# B&R Automation Studio project MotionTestBenchMaster (part 6)

#### SwChg.st - Monitor and write into the user logger the canges of the software objects
```iecst
(********************************************************************
 * COPYRIGHT --
 ********************************************************************
 * Library: Powertoys
 * File: swChg.st
 * Author: Massimo Gibertini
 * Created: August 07, 2014
 ********************************************************************
 * Implementation of library Powertoys
 ********************************************************************)

(* Monitor and write into the user logger the canges of the software objects *)
FUNCTION_BLOCK SwChg

	IF (enable = TRUE) THEN
		customEntry.logLevel 		:= logLevel;
		waitWrite.PT				:= T#10m;

		CASE step OF

			0:
				(* Getting the software list *)
				busy			:= TRUE;
				searching		:= FALSE;
				writingLog		:= FALSE;
				waiting			:= FALSE;
				scan			:= TRUE;
				error			:= FALSE;
				errorID			:= ERR_FUB_BUSY;

				CASE substep OF

					0:
						memset(ADR(tempModule),0,SIZEOF(tempModule));
						memset(ADR(iActList),0,SIZEOF(iActList));
						memset(ADR(iOldList),0,SIZEOF(iOldList));

						(* Checking if the swList temporary data object exist in the userRam or not*)
						datObjInfo_0.pName 	:= ADR(swListTempDataObjName);
						datObjInfo_0.enable	:= TRUE;
						substep 			:= 1;

					1:
						datObjInfo_0();
						IF (datObjInfo_0.status = doERR_MODULNOTFOUND) THEN
							(* Temporary data object not found *)
							swListTempID	:= 0;
							substep			:= 5;
						ELSIF (datObjInfo_0.status = ERR_OK) THEN
							(* Data object found *)
							swListTempID	:= datObjInfo_0.ident;
							//substep			:= 2;
							substep			:= 5;
						ELSIF (datObjInfo_0.status <> ERR_OK) AND (datObjInfo_0.status <> doERR_MODULNOTFOUND) AND (datObjInfo_0.status <> ERR_FUB_BUSY) THEN
							errorID			:= datObjInfo_0.status;
							errorStep		:= step;
							errorSubStep	:= substep;
							step 			:= 200;
							substep			:= 0;
						END_IF;

					2:
						datObjInfo_0.enable	:= FALSE;
						datObjInfo_0();
						IF (datObjInfo_0.status = ERR_FUB_ENABLE_FALSE) THEN
							substep			:= 3;
						END_IF;

					3:
						(* Delete the temporary data object *)
						datObjDelete_0.ident	:= swListTempID;
						datObjDelete_0.enable	:= TRUE;
						substep					:= 4;

					4:
						datObjDelete_0();
						IF (datObjDelete_0.status = ERR_OK) THEN
							substep			:= 5;
							swListTempID	:= 0;
						ELSIF (datObjDelete_0.status <> ERR_OK) AND (datObjDelete_0.status <> ERR_FUB_BUSY) THEN
							errorID			:= datObjDelete_0.status;
							errorStep		:= step;
							errorSubStep	:= substep;
							step 			:= 200;
							substep			:= 0;
						END_IF;

					5:
						(* Disable fub *)
						datObjDelete_0.enable	:= FALSE;
						datObjDelete_0();
						datObjInfo_0.enable	:= FALSE;
						datObjInfo_0();
						IF (datObjDelete_0.status = ERR_FUB_ENABLE_FALSE) AND (datObjInfo_0.status = ERR_FUB_ENABLE_FALSE) THEN
							substep				:= 6;
						END_IF;

					6:
						(* temporary data object not present or deleted *)
						(* Checking if the swList data object exist or not *)
						datObjInfo_0.pName 	:= ADR(swListDatObjName);
						datObjInfo_0.enable	:= TRUE;
						datObjInfo_0();
						IF (datObjInfo_0.status <> ERR_FUB_BUSY) AND (datObjInfo_0.status <> ERR_FUB_ENABLE_FALSE) THEN
							substep := 7;
						END_IF;

					7:
						datObjInfo_0();
						IF (datObjInfo_0.status = doERR_MODULNOTFOUND) THEN
							(* Data object not found *)
							swListID		:= 0;
							substep			:= 100;
						ELSIF (datObjInfo_0.status = doERR_CHECKSUM_WARNING) THEN
							swListID		:= datObjInfo_0.ident;
							substep			:= 10;
						ELSIF (datObjInfo_0.status = ERR_OK) THEN
							(* Data object found *)
							swListID		:= datObjInfo_0.ident;
							IF (swListTempID = 0) THEN
								substep			:= 50;
							ELSE
								substep 		:= 150;
							END_IF;

						ELSIF (datObjInfo_0.status <> ERR_OK) AND (datObjInfo_0.status <> doERR_CHECKSUM_WARNING) AND (datObjInfo_0.status <> doERR_MODULNOTFOUND) AND (datObjInfo_0.status <> ERR_FUB_BUSY) THEN
							errorID			:= datObjInfo_0.status;
							errorStep		:= step;
							errorSubStep	:= substep;
							step 			:= 200;
							substep			:= 0;
						END_IF;

					(* Data object damaged, deleting *)
					10:
						datObjInfo_0.enable	:= FALSE;
						datObjInfo_0();
						IF (datObjInfo_0.status = ERR_FUB_ENABLE_FALSE) THEN
							substep			:= 11;
						END_IF;

					11:
						datObjDelete_0.ident	:= swListID;
						datObjDelete_0.enable	:= TRUE;
						datObjDelete_0();
						IF (datObjDelete_0.status <> ERR_FUB_BUSY) AND (datObjDelete_0.status <> ERR_FUB_ENABLE_FALSE) THEN
							substep 				:= 12;
						END_IF;

					12:
						datObjDelete_0();
						IF (datObjDelete_0.status = ERR_OK) THEN
							substep				:= 13;
						ELSIF (datObjDelete_0.status <> ERR_OK) AND (datObjDelete_0.status <> ERR_FUB_BUSY) THEN
							errorID				:= datObjDelete_0.status;
							errorStep			:= step;
							errorSubStep		:= substep;
							step 				:= 200;
							substep				:= 0;
						END_IF;

					13:
						datObjDelete_0.enable	:= FALSE;
						datObjDelete_0();
						IF (datObjDelete_0.status = ERR_FUB_ENABLE_FALSE) THEN
							(* No existing data object *)
							substep 			:= 100;
							swListID 			:= 0;
						END_IF;

					50:
						(* swList data object present, copy to DRam *)
						datObjInfo_0.enable			:= FALSE;
						datObjCopy_0.ident 			:= swListID;
						datObjCopy_0.pNameTarget 	:= ADR(swListTempDataObjName);
						datObjCopy_0.MemTypeTarget	:= doTEMP;
						datObjCopy_0.enable			:= TRUE;
						datObjCopy_0();
						substep := 51;

					51:
						datObjCopy_0();
						IF (datObjCopy_0.status = ERR_OK) THEN
							substep 				:= 52;
							swListTempID			:= datObjCopy_0.identNew;
						ELSIF (datObjCopy_0.status <> ERR_OK) AND (datObjCopy_0.status <> ERR_FUB_BUSY) THEN
							errorID					:= datObjCopy_0.status;
							errorStep				:= step;
							errorSubStep			:= substep;
							step 					:= 200;
							substep					:= 0;
						END_IF;

					52:
						datObjCopy_0.enable			:= FALSE;
						datObjCopy_0();
						IF (datObjCopy_0.status = ERR_FUB_ENABLE_FALSE) THEN
							(* Temporary Data object recovered succesfully *)
							substep					:= 150;

						END_IF;

					100:
						(* Creating the temporary data object*)
						IF (swListTempID = 0) THEN
							datObjInfo_0.enable		:= FALSE;
							datObjCreate_0.grp		:= 0;
							datObjCreate_0.pName	:= ADR(swListTempDataObjName);
							datObjCreate_0.len		:= SIZEOF(iActList);
							datObjCreate_0.MemType	:= doTEMP;
							datObjCreate_0.Option	:= doNO_CS;
							datObjCreate_0.pCpyData	:= ADR(iActList);
							datObjCreate_0.enable	:= TRUE;
							datObjCreate_0();
							substep					:= 101;
						ELSE
							substep					:= 110;
						END_IF;

					101:
						datObjCreate_0();
						IF (datObjCreate_0.status = ERR_OK) THEN
							substep				:= 102;
							swListTempID		:= datObjCreate_0.ident;
							newSwListT			:= TRUE;
						ELSIF (datObjCreate_0.status <> ERR_OK) AND (datObjCreate_0.status <> ERR_FUB_BUSY) THEN
							errorID				:= datObjCreate_0.status;
							errorStep			:= step;
							errorSubStep		:= substep;
							step 				:= 200;
							substep				:= 0;
						END_IF;

					102:
						datObjCreate_0.enable	:= FALSE;
						datObjCreate_0();
						IF (datObjCreate_0.status = ERR_FUB_ENABLE_FALSE) THEN
							substep				:= 110;

						END_IF;

					110:
						(* Creating the cf data object*)
						datObjCreate_0.grp		:= 0;
						datObjCreate_0.pName	:= ADR(swListDatObjName);
						datObjCreate_0.len		:= SIZEOF(iOldList);
						datObjCreate_0.MemType	:= doUSRROM;
						datObjCreate_0.Option	:= 0;
						datObjCreate_0.pCpyData	:= ADR(iOldList);
						datObjCreate_0.enable	:= TRUE;
						substep					:= 112;

					112:
						datObjCreate_0();
						IF (datObjCreate_0.status = ERR_OK) THEN
							substep					:= 113;
							swListID				:= datObjCreate_0.ident;
							datObjCreate_0.enable	:= FALSE;
						ELSIF (datObjCreate_0.status <> ERR_OK) AND (datObjCreate_0.status <> ERR_FUB_BUSY) THEN
							errorID					:= datObjCreate_0.status;
							errorStep				:= step;
							errorSubStep			:= substep;
							step 					:= 200;
							substep					:= 0;
						END_IF;

					113:
						datObjCreate_0.enable		:= FALSE;
						datObjCreate_0();
						IF (datObjCreate_0.status = ERR_FUB_ENABLE_FALSE) AND newSwListT THEN
							substep					:= 200;
							oldListElements			:= 0;
						ELSIF (datObjCreate_0.status = ERR_FUB_ENABLE_FALSE) AND NOT (newSwListT) THEN
							substep					:= 150;
							oldListElements			:= 0;
						END_IF;

					150:
						(* Loading the existing temporary data object *)
						datObjRead_0.ident			:= swListTempID;
						datObjRead_0.Offset			:= 0;
						datObjRead_0.pDestination	:= ADR(iOldList);
						datObjRead_0.len			:= SIZEOF(iOldList);
						datObjRead_0.enable			:= TRUE;
						datObjRead_0();
						substep						:= 151;

					151:

						datObjRead_0();
						IF (datObjRead_0.status = ERR_OK) THEN
							substep					:= 152;
						ELSIF (datObjRead_0.status <> ERR_OK) AND (datObjRead_0.status <> ERR_FUB_BUSY)	THEN
							errorID					:= datObjRead_0.status;
							errorStep				:= step;
							errorSubStep			:= substep;
							step 					:= 200;
							substep					:= 0;
						END_IF;

					152:
						datObjRead_0.enable			:= FALSE;
						datObjRead_0();
						IF (datObjRead_0.status = ERR_FUB_ENABLE_FALSE) THEN
							oldListElements 		:= 0;
							substep 				:= 153;
						END_IF;

					153:
						(* Listing the number of entries in the old list *)
						memset(ADR(tempString),0,SIZEOF(tempString));
						memcpy(ADR(tempString),ADR(iOldList[oldListElements].module.name[0]),SIZEOF(iOldList[oldListElements].module.name));
						IF (tempString <> '') THEN
							oldListElements := oldListElements + 1;
						ELSE
							substep 		:= 200;
						END_IF;

					200:
						(* Cleaning the memory of the actual list *)
						(* Listing all the software objects *)
						memset(ADR(iActList),0,SIZEOF(iActList));
						mo_prev_index 	:= 16#FFFF;
						mo_index 		:= 0;
						nrChanges 		:= 0;
						substep			:= 201;

					201:
						(* Listing all the software objects element *)
						memset(ADR(tempModule), 0, SIZEOF(tempModule));
						MO_list(mo_prev_index, ADR(mo_index),ADR(tempModule));

						IF (tempModule.type <> 0) AND ((tempModule.type = CST_configOBJ)	OR
							(tempModule.type = CST_cycOBJ)		OR
							(tempModule.type = CST_fwOBJ)		OR
							(tempModule.type = CST_hwOBJ)		OR
							(tempModule.type = CST_ncOBJ)		OR
							(tempModule.type = CST_sysOBJ))		THEN

							(* Valid system object *)
							MO_ver(ADR(tempModule.name),0,ADR(iActList[nrChanges].version));
							memcpy(ADR(iActList[nrChanges].module.name[0]),ADR(tempModule.name[0]), SIZEOF(tempModule.name));

							iActList[nrChanges].module.grp		:= tempModule.grp;
							iActList[nrChanges].module.memtype	:= tempModule.memtype;
							iActList[nrChanges].module.reserve 	:= tempModule.reserve;
							iActList[nrChanges].module.state	:= tempModule.state;
							iActList[nrChanges].module.type		:= tempModule.type;

							nrChanges							:= nrChanges + 1;
							substep 							:= 202;
						ELSE
							substep 							:= 202;
						END_IF;

					202:
						(* Checking if I have finished to scan *)

						IF (mo_prev_index = mo_index) OR (nrChanges = iMaxEntries) THEN
							substep 		:= 203;
						ELSE
							mo_prev_index	:= mo_index;
							substep 		:= 201;
						END_IF;

					203:
						(* Software list complete *)
						actListElements 	:= nrChanges;
						step 				:= 1;
						substep 			:= 0;

				END_CASE;

			1:
				(* Searching for modified software objects *)
				busy			:= TRUE;
				searching		:= TRUE;
				writingLog		:= FALSE;
				waiting			:= FALSE;
				scan			:= FALSE;
				error			:= FALSE;
				errorID			:= ERR_FUB_BUSY;

				CASE substep OF
					0:
						(* Software list complete, comparing memory area *)
						IF (memcmp(ADR(iActList), ADR(iOldList), SIZEOF(iActList)) = 0) THEN

							(* No software changes *)
							substep	:= 0;
							step	:= 20;

						ELSE

							(* There are some changes *)
							substep		:= 1;
							cnt			:= 0;
							nrChanges	:= 0;
							oldSubStep	:= 0;
						END_IF;

					1:
						(* Trying to find the module in the same position of the old array *)
						(* First speed up improvement *)
						IF ((memcmp(ADR(iActList[nrChanges].module.name[0]), ADR(iOldList[nrChanges].module.name[0]), SIZEOF(iOldList[nrChanges].module.name)) = 0)
							AND (cnt < oldListElements) AND (nrChanges < actListElements)) THEN

							(* Module found *)
							IF (memcmp(ADR(iActList[nrChanges]),ADR(iOldList[nrChanges]),SIZEOF(iOldList[nrChanges])) = 0) THEN

								(* The module are the same *)
								nrChanges	:= nrChanges + 1;
								cnt			:= 0;
							ELSE

								(* The module is modified *)
								substep 	:= 10;
								step		:= 10;

							END_IF;

						ELSE
							(* Module not found *)
							substep 	:= 10;

						END_IF;

					10:
						(* Comparing the all elements of the iActList with all the elements of iOldList to find if the element exist or not *)
						IF (memcmp(ADR(iActList[nrChanges].module.name[0]), ADR(iOldList[cnt].module.name[0]), SIZEOF(iOldList[cnt].module.name)) <> 0) AND (nrChanges < actListElements) THEN
							IF (cnt < oldListElements)  THEN
								(* Module not found *)
								cnt 		:= cnt + 1;

							ELSIF (cnt >= oldListElements)  THEN

								(* New software module *)
								substep		:= 20;
								step		:= 10;
							END_IF;

						ELSIF ((memcmp(ADR(iActList[nrChanges].module.name[0]), ADR(iOldList[cnt].module.name[0]), SIZEOF(iOldList[cnt].module.name)) = 0)
								AND (cnt < oldListElements) AND (nrChanges < actListElements)) THEN

							(* Module found *)
							IF (memcmp(ADR(iActList[nrChanges]),ADR(iOldList[cnt]),SIZEOF(iOldList[cnt])) = 0) THEN

								(* The module are the same *)
								nrChanges	:= nrChanges + 1;
								cnt			:= 0;
								substep 	:= 1;
							ELSE

								(* The module is modified *)
								substep 	:= 10;
								step		:= 10;
							END_IF;

						ELSIF (nrChanges >= actListElements) THEN

							(* Search finished, checking the removed objects *)
							substep			:= 2;
							cnt 			:= 0;
							nrChanges 		:= 0;
						END_IF;

					2:
						(* Trying to find the module in the same position of the old array *)
						(* Second speed up improvement *)
						IF ((memcmp(ADR(iActList[cnt].module.name[0]), ADR(iOldList[cnt].module.name[0]), SIZEOF(iOldList[cnt].module.name)) = 0)
							AND (cnt < oldListElements) AND (nrChanges < actListElements)) THEN

							(* Module found *)
							cnt				:= cnt + 1;
							nrChanges		:= 0;

						ELSE
							(* Module not found *)
							nrChanges		:= 0;
							substep 	:= 20;
						END_IF

					20:
						(* Checking if there are any removed software object *)
						IF (memcmp(ADR(iActList[nrChanges].module.name[0]), ADR(iOldList[cnt].module.name[0]), SIZEOF(iOldList[cnt].module.name)) <> 0) AND (oldListElements <> 0) AND (cnt < oldListElements) THEN

							IF  (nrChanges < actListElements) THEN

								(* Module not found *)
								nrChanges	:= nrChanges + 1;

							ELSIF (nrChanges >= actListElements) THEN

								(* SW module removed *)
								substep 	:= 0;
								step		:= 10;
							END_IF;

						ELSIF ((memcmp(ADR(iActList[nrChanges].module.name[0]), ADR(iOldList[cnt].module.name[0]), SIZEOF(iOldList[cnt].module.name)) = 0)
							AND (cnt < oldListElements) AND (nrChanges < actListElements)) THEN

							(* Module found *)
							cnt				:= cnt + 1;
							substep 		:= 2;
							nrChanges		:= 0;

						ELSIF (cnt >= oldListElements) THEN

							(* Search finished *)
							step			:= 10;
							substep 		:= 30;
							cnt				:= 0;
							nrChanges		:= 0;
						END_IF;

				END_CASE;

			10:
				(* Writing informations into the logger and data object *)
				busy 			:= TRUE;
				searching 		:= FALSE;
				writingLog		:= TRUE;
				waiting 		:= FALSE;
				scan			:= FALSE;
				error			:= FALSE;
				errorID			:= ERR_FUB_BUSY;

				CASE substep OF

					0:
						(* Removed software module *)
						memset(ADR(tempString),0,SIZEOF(tempString));
						tempString	:= 'REMOVED SW MODULE: ';
						memcpy(ADR(tempString)+LEN(tempString),ADR(iOldList[cnt].module.name[0]), SIZEOF(iOldList[cnt].module.name));
						substep		:= 1;

					1:
						(* Writing into the logger *)
						customEntry.adr_string 		:= ADR(tempString);
						customEntry.errorNum 		:= LOG_SW_OBJ_CHG;
						writeDiff.adrCustomEntry 	:= ADR(customEntry);
						writeDiff.enable 			:= TRUE;
						substep 					:= 2;

					2:

						IF (writeDiff.done = TRUE) THEN
							substep			:= 3;
						ELSIF (writeDiff.error) THEN
							errorID			:= writeDiff.errorID;
							errorStep		:= step;
							errorSubStep	:= substep;
							step 			:= 200;
							substep			:= 0;
						END_IF;

					3:
						writeDiff.enable	:= FALSE;
						IF (writeDiff.errorID = ERR_FUB_ENABLE_FALSE) THEN
							cnt				:= cnt + 1;
							nrChanges		:= 0;
							step			:= 1;
							substep			:= 2;
						END_IF;

					10:
						(* Modified software module *)
						memset(ADR(tempString),0,SIZEOF(tempString));
						tempString	:= 'MODIFIED SW MODULE: ';
						memcpy(ADR(tempString)+LEN(tempString),ADR(iActList[nrChanges].module.name[0]), SIZEOF(iActList[nrChanges].module.name));
						substep		:= 11;

					11:
						(* Writing into the logger *)
						customEntry.adr_string 		:= ADR(tempString);
						customEntry.errorNum 		:= LOG_SW_OBJ_CHG;
						writeDiff.adrCustomEntry 	:= ADR(customEntry);
						writeDiff.enable 			:= TRUE;
						substep 					:= 12;

					12:

						IF (writeDiff.done = TRUE) THEN
							substep			:= 13;
						ELSIF (writeDiff.error) THEN
							errorID			:= writeDiff.errorID;
							errorStep		:= step;
							errorSubStep	:= substep;
							step 			:= 200;
							substep			:= 0;
						END_IF;

					13:
						writeDiff.enable	:= FALSE;
						IF (writeDiff.errorID = ERR_FUB_ENABLE_FALSE) THEN
							cnt				:= 0;
							nrChanges		:= nrChanges + 1;
							substep			:= 1;
							step			:= 1;
						END_IF;

					20:
						(* New software module *)
						memset(ADR(tempString),0,SIZEOF(tempString));
						tempString	:= 'NEW SW MODULE: ';
						memcpy(ADR(tempString)+LEN(tempString),ADR(iActList[nrChanges].module.name[0]), SIZEOF(iActList[nrChanges].module.name));
						substep		:= 21;

					21:
						(* Writing into the logger *)
						customEntry.adr_string 		:= ADR(tempString);
						customEntry.errorNum 		:= LOG_SW_OBJ_NEW;
						writeDiff.adrCustomEntry 	:= ADR(customEntry);
						writeDiff.enable 			:= TRUE;
						substep						:= 22;

					22:
						IF (writeDiff.done = TRUE) THEN
							substep			:= 23;
						ELSIF (writeDiff.error) THEN
							errorID			:= writeDiff.errorID;
							errorStep		:= step;
							errorSubStep	:= substep;
							step 			:= 200;
							substep			:= 0;
						END_IF;

					23:
						writeDiff.enable	:= FALSE;
						IF (writeDiff.errorID = ERR_FUB_ENABLE_FALSE) THEN
							cnt				:= 0;
							nrChanges		:= nrChanges + 1;
							substep			:= 1;
							step			:= 1;
						END_IF;

					30:
						(* Writing temporary data object *)
						datObjWrite_0.ident		:= swListTempID;
						datObjWrite_0.len		:= SIZEOF(iActList);
						datObjWrite_0.Offset	:= 0;
						datObjWrite_0.pSource	:= ADR(iActList);
						datObjWrite_0.enable	:= TRUE;
						datObjWrite_0();
						substep					:= 31;

					31:
						datObjWrite_0();
						IF (datObjWrite_0.status = ERR_OK) THEN
							substep 				:= 50;
							waitWrite.IN 			:= TRUE;
							datObjWrite_0.enable 	:= FALSE;
						ELSIF (datObjWrite_0.status <> ERR_OK) AND (datObjWrite_0.status <> ERR_FUB_BUSY) THEN
							errorID					:= datObjWrite_0.status;
							errorStep				:= step;
							errorSubStep			:= substep;
							step 					:= 200;
							substep					:= 0;
						END_IF;

					40:
						(* Writing cf data object *)
						datObjWrite_0.ident			:= swListID;
						datObjWrite_0.len			:= SIZEOF(iActList);
						datObjWrite_0.Offset		:= 0;
						datObjWrite_0.pSource		:= ADR(iActList);
						datObjWrite_0.enable		:= TRUE;
						datObjWrite_0();
						substep						:= 41;
					41:
						datObjWrite_0();
						IF (datObjWrite_0.status = ERR_OK) THEN
							substep 				:= 50;
							waitWrite.IN 			:= FALSE;
							datObjWrite_0.enable 	:= FALSE;
						ELSIF (datObjWrite_0.status <> ERR_OK) AND (datObjWrite_0.status <> ERR_FUB_BUSY) THEN
							errorID					:= datObjWrite_0.status;
							errorStep				:= step;
							errorSubStep			:= substep;
							step 					:= 200;
							substep					:= 0;
						END_IF;

					50:
						(* Copy the actual list into the old list *)
						memcpy(ADR(iOldList), ADR(iActList), SIZEOF(iActList));
						memset(ADR(tempString),0,SIZEOF(tempString));
						substep := 0;
						step 	:= 20;
				END_CASE;

			20:
				(* Waiting step *)
				busy 			:= TRUE;
				searching 		:= FALSE;
				writingLog		:= FALSE;
				waiting 		:= TRUE;
				scan			:= FALSE;
				error			:= FALSE;
				errorID			:= ERR_FUB_BUSY;

				CASE substep OF
					0:
						(* No software changes *)
						refresh.PT := refreshTime;
						refresh.IN := TRUE;

						IF refresh.Q THEN
							substep := 1;
						END_IF;

					1:
						(* Refresh time elapsed *)
						IF (waitWrite.Q) THEN
							step 	:= 10;
							substep := 40;
						ELSE
							refresh.IN := FALSE;
							step 	:= 0;
							substep := 152;
						END_IF;

				END_CASE;

			200:
				(* Error state resetting all the used function block *)
				writeDiff.enable		:= FALSE;
				refresh.IN 				:= FALSE;
				waitWrite.IN			:= FALSE;
				datObjWrite_0.enable	:= FALSE;
				datObjInfo_0.enable		:= FALSE;
				datObjDelete_0.enable	:= FALSE;
				datObjRead_0.enable		:= FALSE;
				datObjCreate_0.enable	:= FALSE;
				datObjCopy_0.enable		:= FALSE;

				(* Updating the status *)
				busy			:= FALSE;
				searching		:= FALSE;
				writingLog		:= FALSE;
				waiting			:= FALSE;
				scan			:= FALSE;
				error			:= TRUE;
		END_CASE;

	ELSE

		mo_prev_index 	:= 16#FFFF;
		mo_index 		:= 0;
		cnt 			:= 0;
		nrChanges 		:= 0;
		substep			:= 0;
		step			:= 0;
		errorSubStep	:= 0;
		errorStep		:= 0;
		oldSubStep		:= 0;

		oldListElements := 0;
		actListElements	:= 0;

		error			:= TRUE;
		errorID			:= ERR_FUB_ENABLE_FALSE;
		busy			:= FALSE;
		searching		:= FALSE;
		writingLog		:= FALSE;
		waiting			:= FALSE;
		scan			:= FALSE;
		newSwListT		:= FALSE;
		(* Resetting all the used function block *)
		writeDiff.enable		:= FALSE;
		refresh.IN 				:= FALSE;
		waitWrite.IN			:= FALSE;
		datObjWrite_0.enable	:= FALSE;
		datObjInfo_0.enable		:= FALSE;
		datObjDelete_0.enable	:= FALSE;
		datObjRead_0.enable		:= FALSE;
		datObjCreate_0.enable	:= FALSE;
		datObjCopy_0.enable		:= FALSE;
	END_IF;

	writeDiff();
	refresh();
	waitWrite();

END_FUNCTION_BLOCK
```

#### LogSupplyEvents.st - Write the power supply events in the specified logger
```iecst
(********************************************************************
 * COPYRIGHT -- Bernecker + Rainer
 ********************************************************************
 * Library: GenUps
 * File: LogSupplyEvents.st
 * Author: gibertinim
 * Created: March 13, 2014
 ********************************************************************
 * Implementation of library GenUps
 ********************************************************************)

(* Write the power supply events in the specified logger *)
FUNCTION_BLOCK LogSupplyEvents

	IF (enable = TRUE) THEN

		CASE step OF

			0:
				pUpsIO ACCESS (ADR_UpsIO);

				errorID 			:=	ERR_FUB_BUSY;
				busy				:=	TRUE;
				error				:=	FALSE;
				noSupply			:= TRUE;
				batteryLow			:= FALSE;
				batteryAlarm		:= FALSE;
				shutdownRequested	:= FALSE;

				IF (customLogEntry_0.errorID = ERR_FUB_ENABLE_FALSE) THEN
					(* The function block started running *)
					step := 1;
				END_IF;

			1:

				memset(ADR(data),0,SIZEOF(data));
				customLogEntry_0.adrCustomEntry	:=	ADR(data);
				memset(ADR(tempString),0,SIZEOF(tempString));
				memset(ADR(tempString2),0,SIZEOF(tempString2));

				IF (pUpsIO.shutdownAlarm = TRUE) THEN
					step := 50;
				ELSE
					step := 51;
				END_IF;

			2:
				(* Waiting for an event *)

				IF 		((pUpsIO.batteryAlarm	= TRUE)		AND	(batteryAlarm		= FALSE))	THEN
					step := 10;
				ELSIF	((pUpsIO.batteryAlarm	= FALSE)	AND	(batteryAlarm		= TRUE))	THEN
					step := 11;
				ELSIF	((pUpsIO.batteryLow		= TRUE)		AND	(batteryLow			= FALSE))	THEN
					step := 20;
				ELSIF	((pUpsIO.batteryLow		= FALSE)	AND	(batteryLow			= TRUE))	THEN
					step := 21;
				ELSIF	((pUpsIO.noPowerSupply	= TRUE)		AND (noSupply			= FALSE))	THEN
					step := 30;
				ELSIF	((pUpsIO.noPowerSupply	= FALSE)	AND (noSupply			= TRUE))	THEN
					step := 31;
				ELSIF (pUpsIO.shutdownReq		= TRUE)		AND	(shutdownRequested	= FALSE)	THEN
					step := 40;
				ELSIF(	(pUpsIO.batteryAlarm	= FALSE)	AND	(batteryAlarm		= FALSE)	AND
						(pUpsIO.batteryLow		= FALSE)	AND	(batteryLow			= FALSE)	AND
						(pUpsIO.noPowerSupply	= FALSE)	AND (noSupply			= FALSE)	AND
						(pUpsIO.shutdownReq 	= FALSE)	AND (shutdownRequested	= FALSE))	THEN
					upsStatus := ERR_OK;
				ELSIF (	(pUpsIO.shutdownReq 	= FALSE)	AND (shutdownRequested	= TRUE)) THEN
					shutdownRequested := FALSE;
				END_IF;

			10:

				customLogEntry_0.enable 		:= 	TRUE;

				data.errorNum		:= ERR_UPS_BATTERY_FAULT;
				data.adr_string		:= ADR('UPS BATTERY FAULT');
				data.logLevel		:= arEVENTLOG_SEVERITY_WARNING;
				batteryAlarm		:= TRUE;
				upsStatus			:= ERR_UPS_BATTERY_FAULT;
				(* Waiting until the log is written succesfully *)
				IF (customLogEntry_0.errorID = ERR_OK) THEN
					(* Log entry written succesfully*)
					step 					:= 101;
					customLogEntry_0.enable := 	FALSE;
				ELSIF ((customLogEntry_0.errorID <> ERR_FUB_BUSY) AND (customLogEntry_0.errorID <> ERR_OK)AND (customLogEntry_0.errorID <> ERR_FUB_ENABLE_FALSE)) THEN
					(* Error occured while saving the logger *)
					errorStep	:= 10;
					errorID		:= customLogEntry_0.errorID;
					error		:= TRUE;
					step		:= 200;
				END_IF;

			11:
				(* Battery alarm recovered *)

				customLogEntry_0.enable := 	TRUE;
				data.errorNum			:= ERR_UPS_BATTERY_OK;

				data.adr_string	:= ADR('UPS BATTERY FAULT RECOVERED');
				data.logLevel	:= arEVENTLOG_SEVERITY_INFO;
				batteryAlarm	:= FALSE;
				(* Waiting until the log is written succesfully *)

				IF (customLogEntry_0.errorID = ERR_OK) THEN
					(* Log entry written succesfully*)
					step 					:= 101;
					customLogEntry_0.enable := FALSE;
				ELSIF ((customLogEntry_0.errorID <> ERR_FUB_BUSY) AND customLogEntry_0.errorID <> ERR_OK)AND (customLogEntry_0.errorID <> ERR_FUB_ENABLE_FALSE) THEN
					(* Error occured while saving the logger *)
					errorStep	:= 11;
					errorID		:= customLogEntry_0.errorID;
					error		:= TRUE;
					step		:= 200;
				END_IF;

			20:

				(* Battery low *)

				customLogEntry_0.enable 		:= 	TRUE;
				data.errorNum		:= ERR_UPS_BATTERY_LOW;
				data.adr_string		:= ADR('UPS BATTERY LOW');
				data.logLevel		:= arEVENTLOG_SEVERITY_WARNING;
				batteryLow			:= TRUE;
				upsStatus			:= ERR_UPS_BATTERY_LOW;
				(* Waiting until the log is written succesfully *)
				IF (customLogEntry_0.errorID = ERR_OK) THEN
					(* Log entry written succesfully*)
					step 					:= 101;
					customLogEntry_0.enable := FALSE;
				ELSIF ((customLogEntry_0.errorID <> ERR_FUB_BUSY) AND (customLogEntry_0.errorID <> ERR_OK)AND (customLogEntry_0.errorID <> ERR_FUB_ENABLE_FALSE)) THEN
					(* Error occured while saving the logger *)
					errorStep	:= 20;
					errorID		:= customLogEntry_0.errorID;
					error		:= TRUE;
					step		:= 200;
				END_IF;

			21:
				(* Battery recharged *)

				customLogEntry_0.enable 		:= 	TRUE;

				data.errorNum		:= ERR_UPS_BATTERY_CHARGED;
				data.adr_string		:= ADR('UPS BATTERY CHARGED');
				data.logLevel		:= arEVENTLOG_SEVERITY_INFO;
				batteryLow			:= FALSE;
				(* Waiting until the log is written succesfully *)

				IF (customLogEntry_0.errorID = ERR_OK) THEN
					(* Log entry written succesfully*)
					step 					:= 2;
					customLogEntry_0.enable := FALSE;
				ELSIF ((customLogEntry_0.errorID <> ERR_FUB_BUSY) AND (customLogEntry_0.errorID <> ERR_OK)AND (customLogEntry_0.errorID <> ERR_FUB_ENABLE_FALSE)) THEN
					(* Error occured while saving the logger *)
					errorStep	:= 21;
					errorID		:= customLogEntry_0.errorID;
					error		:= TRUE;
					step		:= 200;
				END_IF;

			30:

				(* Lost Power supply *)

				data.errorNum			:= ERR_UPS_NO_SUPPLY;
				data.adr_string			:= ADR('UPS NO POWER SUPPLY');
				data.logLevel			:= arEVENTLOG_SEVERITY_WARNING;
				noSupply				:= TRUE;
				upsStatus				:= ERR_UPS_NO_SUPPLY;
				customLogEntry_0.enable := 	TRUE;
				(* Waiting until the log is written succesfully *)
				IF (customLogEntry_0.errorID = ERR_OK) THEN
					(* Log entry written succesfully*)
					step 					:= 101;
					customLogEntry_0.enable := FALSE;
				ELSIF ((customLogEntry_0.errorID<> ERR_FUB_BUSY) AND (customLogEntry_0.errorID <> ERR_OK)AND (customLogEntry_0.errorID <> ERR_FUB_ENABLE_FALSE)) THEN
					(* Error occured while saving the logger *)
					errorStep	:= 30;
					errorID		:= customLogEntry_0.errorID;
					error		:= TRUE;
					step		:= 200;
				END_IF;

			31:
				(* Power supply ok *)

				customLogEntry_0.enable 		:= 	TRUE;

				data.errorNum		:= ERR_UPS_SUPPLY_BACK;
				data.adr_string		:= ADR('UPS POWER SUPPLY OK');
				data.logLevel		:= arEVENTLOG_SEVERITY_INFO;
				noSupply			:= FALSE;
				(* Waiting until the log is written succesfully *)
				IF (customLogEntry_0.errorID = ERR_OK) THEN
					(* Log entry written succesfully*)
					step 					:= 101;
					customLogEntry_0.enable := FALSE;
				ELSIF ((customLogEntry_0.errorID <> ERR_FUB_BUSY) AND (customLogEntry_0.errorID <> ERR_OK) AND (customLogEntry_0.errorID <> ERR_FUB_ENABLE_FALSE)) THEN
					(* Error occured while saving the logger *)
					errorStep	:= 31;
					errorID		:= customLogEntry_0.errorID;
					error		:= TRUE;
					step		:= 200;
				END_IF;

			40:
				(* Shutdown request *)

				customLogEntry_0.enable 		:= 	TRUE;

				data.errorNum		:= ERR_UPS_SHUTDOWN_REQ;
				data.adr_string		:= ADR('UPS SHUTDOWN REQUEST');
				data.logLevel		:= arEVENTLOG_SEVERITY_INFO;
				shutdownRequested	:= TRUE;
				upsStatus			:= ERR_UPS_SHUTDOWN_REQ;
				(* Waiting until the log is written succesfully *)
				IF (customLogEntry_0.errorID = ERR_OK) THEN
					(* Log entry written succesfully*)
					step 					:= 101;
					customLogEntry_0.enable := FALSE;
				ELSIF ((customLogEntry_0.errorID <> ERR_FUB_BUSY) AND (customLogEntry_0.errorID <> ERR_OK) AND (customLogEntry_0.errorID <> ERR_FUB_ENABLE_FALSE)) THEN
					(* Error occured while saving the logger *)
					errorStep	:= 40;
					errorID		:= customLogEntry_0.errorID;
					error		:= TRUE;
					step		:= 200;
				END_IF;

			50:
				(* Writing the total power off time to the logger *)
				(* Shutdown request *)
				itoa(pUpsIO.powerOffTime, ADR(tempString));
				tempString2 := 'UPS SHUTDOWN TIME ';
				strcat(ADR(tempString2), ADR(tempString));
				strcat(ADR(tempString2), ADR('s'));

				customLogEntry_0.enable 		:= 	TRUE;
				data.errorNum					:= ERR_UPS_SHUTDOWN_TIME;
				data.adr_string					:= ADR(tempString2);
				data.logLevel					:= arEVENTLOG_SEVERITY_INFO;
				shutdownRequested				:= TRUE;
				upsStatus						:= ERR_UPS_SHUTDOWN_REQ;

				(* Waiting until the log is written succesfully *)
				IF (customLogEntry_0.errorID = ERR_OK) THEN
					(* Log entry written succesfully*)
					step 					:= 51;
					customLogEntry_0.enable := FALSE;
				ELSIF ((customLogEntry_0.errorID <> ERR_FUB_BUSY) AND (customLogEntry_0.errorID <> ERR_OK) AND (customLogEntry_0.errorID <> ERR_FUB_ENABLE_FALSE)) THEN
					(* Error occured while saving the logger *)
					errorStep	:= 50;
					errorID		:= customLogEntry_0.errorID;
					error		:= TRUE;
					step		:= 200;
				END_IF;

			51:

				(* Identifier obtained succesfully *)
				IF (pUpsIO.noPowerSupply = TRUE) THEN
					step := 30;
				ELSE
					step := 31;
				END_IF;

			100:
				(* Waiting until the log is written succesfully *)
				IF (customLogEntry_0.errorID = ERR_OK) THEN
					(* Log entry written succesfully*)
					step := 101;

				ELSIF ((customLogEntry_0.errorID <> ERR_FUB_BUSY) AND (customLogEntry_0.errorID <> ERR_OK) AND (customLogEntry_0.errorID <> ERR_FUB_ENABLE_FALSE)) THEN
					(* Error occured while saving the logger *)
					errorStep	:= 100;
					errorID		:= customLogEntry_0.errorID;
					error		:= TRUE;
					step		:= 200;
				END_IF

			101:
			(* Disabling the function block *)
				IF (customLogEntry_0.errorID = ERR_FUB_ENABLE_FALSE) THEN
					memset(ADR(data),0,SIZEOF(data));
					step 			:= 2;
				END_IF;

			200:
			(* Error step *)
				customLogEntry_0.enable	:=	FALSE;

		END_CASE;

	ELSE

		error					:= TRUE;
		errorID					:= ERR_FUB_ENABLE_FALSE;
		customLogEntry_0.enable	:=	FALSE;
		step					:= 0;
		errorStep				:= 0;
		upsStatus				:= ERR_OK;
		noSupply				:= TRUE;
		batteryLow				:= FALSE;
		batteryAlarm			:= FALSE;
		shutdownRequested		:= FALSE;
		busy					:= FALSE;
		memset(ADR(data),0,SIZEOF(data));
	END_IF;

	customLogEntry_0();
END_FUNCTION_BLOCK
```

#### SynchLog.st - Machine synchronization logger
```iecst
(********************************************************************
 * COPYRIGHT --
 ********************************************************************
 * Library: SidelLog
 * File: SynchLog.st
 * Author: Administrator
 * Created: July 15, 2014
 ********************************************************************
 * Implementation of library SidelLog
 ********************************************************************)

(* Machine synchronization logger *)
FUNCTION_BLOCK SynchLog

	IF (enable = TRUE) THEN

		CASE step OF

			0:

				errorID 			:=	ERR_FUB_BUSY;
				busy				:=	TRUE;
				error				:=	FALSE;

				IF (customLogEntry_0.errorID = ERR_FUB_ENABLE_FALSE) THEN
					(* The function block started running *)
					step := 1;
				END_IF;

			1:
				memset(ADR(data),0,SIZEOF(data));

				data.adr_string			:= 	ADR(phasingString);

				customLogEntry_0.adrCustomEntry	:=	(ADR(data));

				rTrig_0.CLK				:=	offsetAcquire;
				customLogEntry_0.enable	:=	FALSE;

				IF rTrig_0.Q	=	TRUE THEN
					step					:=	2;
				END_IF;

			2:
				customLogEntry_0.enable	:=	TRUE;

				data.errorNum	:= LOG_SYNC_AXIS;
				data.logLevel	:= arEVENTLOG_SEVERITY_INFO;

				phasingString	:=	'Homing of Axis ';
				strcat(ADR(phasingString),ADR(axisNameHoming));
				strcat(ADR(phasingString), ADR(' DONE , old position '));
				ftoa(positionMmHoming,ADR(phasingAxisPosition));
				strcat(ADR(phasingString),ADR(phasingAxisPosition));
				strcat(ADR(phasingString), ADR('mm'));

				IF customLogEntry_0.errorID = ERR_OK THEN
					step					:=	10;
					customLogEntry_0.enable	:=	FALSE;
					indexAxis				:=	RAX1;

				ELSIF	((customLogEntry_0.errorID <> ERR_FUB_BUSY) AND (customLogEntry_0.errorID <> ERR_OK)AND (customLogEntry_0.errorID <> ERR_FUB_ENABLE_FALSE)) THEN
					errorStep	:= 	2;
					errorID		:=	customLogEntry_0.errorID;
					error		:=	TRUE;
					step		:=	200;
				END_IF;

			10:
				IF (customLogEntry_0.errorID=ERR_FUB_ENABLE_FALSE) THEN

					step		:=	20;
					indexAxis	:=	RAX1;
					testIndex	:=  RAX1;
				END_IF;

			20:
				IF indexAxis <= AXN THEN

					IF testBit = TRUE THEN

						customLogEntry_0.enable	:=	TRUE;
						data.errorNum	:= LOG_AXIS_POSITION;
						data.logLevel	:= arEVENTLOG_SEVERITY_INFO;

						phasingString	:=	'Position of Axis ';
						strcat(ADR(phasingString),ADR(axisName));
						strcat(ADR(phasingString), ADR(' is '));
						ftoa(positionMm,ADR(phasingAxisPosition));
						strcat(ADR(phasingString),ADR(phasingAxisPosition));
						strcat(ADR(phasingString), ADR('mm'));

						IF customLogEntry_0.errorID = ERR_OK THEN

							customLogEntry_0.enable	:=	FALSE;
							step					:=21;
						ELSIF	((customLogEntry_0.errorID <> ERR_FUB_BUSY) AND (customLogEntry_0.errorID <> ERR_OK)AND (customLogEntry_0.errorID <> ERR_FUB_ENABLE_FALSE)) THEN
							errorStep	:= 20;
							errorID		:= customLogEntry_0.errorID;
							error		:= TRUE;
							step		:=	200;

						END_IF;

					ELSE
						indexAxis	:=	indexAxis+1;
						testIndex	:=	indexAxis;
					END_IF;
				ELSE

					step	:=	1;

				END_IF;
			21:
				IF (customLogEntry_0.errorID=ERR_FUB_ENABLE_FALSE) THEN
					step		:=	20;
					indexAxis	:=	indexAxis+1;
					testIndex	:=	indexAxis;
				END_IF;

			200:
				customLogEntry_0.enable	:=	FALSE;

		END_CASE;

	ELSE

				error					:=	TRUE;
				errorID					:=	ERR_FUB_ENABLE_FALSE;
				customLogEntry_0.enable	:=	FALSE;
				step					:=	0;
				testIndex				:=	0;
				memset(ADR(data),0,SIZEOF(data));
	END_IF;

	customLogEntry_0();
	rTrig_0();

END_FUNCTION_BLOCK
```

### Library Logical/00_AID/Libraries/Sidel_Libraries/Sidel (IEC)
Depends on: LoopConR

#### Sidel.fun - Exported functions and function blocks
```iecst
FUNCTION FC_Parity : BOOL (*TRUE = Even - FALSE = ODD*)
	VAR_INPUT
		IN_Value : DINT;
	END_VAR
END_FUNCTION

FUNCTION_BLOCK AlarmScheduler (*V4.A.A.1.6.13*)
	VAR_INPUT
		AlarmAreaCfg : ARRAY[0..24] OF AlarmAreaCfg_Type;
		AdrAlarm : UDINT;
		AdrAlarmCFG : UDINT;
		AdrAlarmOldStatus : UDINT;
		AdrHMI : UDINT;
	END_VAR
	VAR_OUTPUT
		AlarmAction : ActionSum_Type;
	END_VAR
	VAR_IN_OUT
		FirstAlarmActive : AlarmCFG_Type;
		FirstExternalAlarmActive : AlarmCFG_Type;
		FirstCriticalAlarmActive : AlarmCFG_Type; (*V4.A.A.1.7.0*)
		FirstAlertAlarmActive : AlarmCFG_Type; (*V4.A.A.1.7.0*)
		FirstExtCriticalAlarmActive : AlarmCFG_Type; (*V4.A.A.1.7.0*)
		FirstExtAlertAlarmActive : AlarmCFG_Type; (*V4.A.A.1.7.0*)
		FirstCsAlarmActive : AlarmCFG_Type; (*V4.A.A.1.7.0*)
		FirstCsExtAlarmActive : AlarmCFG_Type; (*V4.A.A.1.7.5a*)
		CriticalAcknoledgeRequest : BOOL;
		AlarmAcknoledgeRequest : BOOL;
	END_VAR
	VAR
		Alarm : REFERENCE TO AlarmCmd_Type;
		AlarmOldStatus : REFERENCE TO BOOL;
		AlarmCFG : REFERENCE TO AlarmCFG_Type;
		HMI : REFERENCE TO BYTE;
		AlarmActionTemp : ActionSum_Type;
		i : UINT;
		x : UINT;
	END_VAR
END_FUNCTION_BLOCK

FUNCTION_BLOCK FirstAlarmCombiner (*V4.A.A.1.6.13*)
	VAR_INPUT
		SkidAlarmFrom : UINT := 1;
		SkidAlarmTo : UINT;
		SkidFirstAlarm : INT;
		SkidFirstExternalAlarm : INT;
		AdrAlarmCFG : UDINT; (*V1.7.4*)
	END_VAR
	VAR_IN_OUT
		FirstAlarmActive : AlarmCFG_Type;
		FirstExternalAlarmActive : AlarmCFG_Type;
	END_VAR
	VAR
		AlarmCFG : REFERENCE TO AlarmCFG_Type; (*V1.7.4*)
	END_VAR
END_FUNCTION_BLOCK

FUNCTION_BLOCK AnalogTotalizer
	VAR_INPUT
		IN_Pulse : BOOL;
		IN_AnalogPV : REAL;
		IN_PulseWeight : REAL;
		IN_ConfigType : USINT; (*Configuaration Time to mapping if analog value is used
(0 = Pulse, 1 = Hours, 2 = Minutes, 3 = Seconds)*)
		IN_Reset : BOOL; (*Reset totalizer*)
	END_VAR
	VAR_IN_OUT
		OUT_TotalCounter : REAL; (*Out Total Counter*)
	END_VAR
	VAR
		RTInfo : RTInfo;
		VAR_AuxPulse : REAL;
		zzEdge00000 : BOOL;
	END_VAR
END_FUNCTION_BLOCK

FUNCTION_BLOCK CyclicActivation
	VAR_INPUT
		IN_CycleTime : TIME;
	END_VAR
	VAR_OUTPUT
		OUT_A : BOOL;
		OUT_B : BOOL;
	END_VAR
	VAR
		TMR_TON_CycleA : TON;
		TMR_TON_CycleB : TON;
		VAR_RtInfo : RTInfo;
		VAR_CycleCounter : REAL;
		VAR_CycleTime : REAL;
		VAR_Cycle : BOOL;
	END_VAR
END_FUNCTION_BLOCK

FUNCTION ComboBoxString : BOOL
	VAR_INPUT
		IN_ElementsStructure : ARRAY[0..19] OF HMI_ComboBoxElements_Type; (*vrma*)
		OUT_ComboString : REFERENCE TO STRING[500];
	END_VAR
	VAR
		VAR_ElementsIndex : USINT;
		VAR_StrIndex : STRING[2];
		VAR_StrComma : STRING[1];
		VAR_StrSemicolun : STRING[1];
	END_VAR
END_FUNCTION

FUNCTION LftConAirPressSp : REAL
	VAR_INPUT
		RcpPressureSp : REAL;
		RcpCanDiameter : REAL;
	END_VAR
	VAR CONSTANT
		CST_PistonDiameterExt : REAL := 40.0; (*[mm]*)
		CST_PistonDiameterInt : REAL := 16.0; (*[mm]*)
		CST_PistonSpringStrengthRse : REAL := 120.0; (*[N]*)
	END_VAR
	VAR
		VAR_PistonSurface : REAL; (*[mm2]*)
		VAR_DeltaPProduct : REAL; (*[N]*)
		VAR_DeltaPrexPist : REAL; (*[bar]*)
		VAR_PbasePiston : REAL; (*[bar]*)
	END_VAR
END_FUNCTION

FUNCTION_BLOCK FB_Blinker
	VAR_INPUT
		IN_Freq : REAL;
	END_VAR
	VAR_OUTPUT
		OUT : BOOL;
	END_VAR
	VAR
		TMR_TON_OnDelay : TON;
		TMR_TON_OffDelay : TON;
		VAR_TimeValue : TIME;
	END_VAR
END_FUNCTION_BLOCK

FUNCTION_BLOCK FB_HMI_ITC_Start
	VAR_IN_OUT
		HMI_Data : HMI_ITC_Data_Type;
		AnalogIndexIn : UINT;
		DigitalIndexIn : UINT;
		AnalogIndexOut : UINT;
		DigitalIndexOut : UINT;
	END_VAR
	VAR
		i : UINT;
	END_VAR
END_FUNCTION_BLOCK

FUNCTION_BLOCK FB_HMI_ITC_DigitalBool
	VAR_INPUT
		IN_Visibility : BOOL;
		IN_ReadOnly : BOOL;
		IN_Wait : BOOL;
		IN_Alarm : BOOL;
		IN_IOType : BOOL; (*0: INPUT 1: OUTPUT*)
		IN_Description : STRING[100];
		IN_HMIAutoForce : BOOL;
	END_VAR
	VAR_OUTPUT
		OUT_Man : BOOL;
		OUT_ManValue : BOOL;
	END_VAR
	VAR_IN_OUT
		ITC_IO : BOOL;
		ITC : BOOL;
		HMI_Data : HMI_ITC_Data_Type;
		HMI_Page : HMI_ITC_Page_Type;
		Index : UINT;
	END_VAR
	VAR
		VAR_Auto : BOOL := TRUE;
		VAR_Man : BOOL := FALSE;
		VAR_PageSwitch : BOOL := TRUE;
		VAR_ProgressiveId : UINT;
		VAR_OldPage : USINT;
		zzEdge00000 : BOOL;
		zzEdge00001 : BOOL;
		zzEdge00002 : BOOL;
		zzEdge00003 : BOOL;
	END_VAR
END_FUNCTION_BLOCK

FUNCTION_BLOCK FB_HMI_ITC_DigitalByte
	VAR_INPUT
		IN_Visibility : BOOL;
		IN_ReadOnly : BOOL;
		IN_Wait : BOOL;
		IN_Alarm : BOOL;
		IN_IOType : BOOL; (*0: INPUT 1: OUTPUT*)
		IN_Description : STRING[100];
		IN_HMIAutoForce : BOOL;
		IN_BitNumber : INT;
	END_VAR
	VAR_OUTPUT
		OUT_Man : BOOL;
		OUT_ManValue : BOOL;
	END_VAR
	VAR_IN_OUT
		ITC_IO : BYTE;
		ITC : BOOL;
		HMI_Data : HMI_ITC_Data_Type;
		HMI_Page : HMI_ITC_Page_Type;
		Index : UINT;
	END_VAR
	VAR
		VAR_Auto : BOOL := TRUE;
		VAR_Man : BOOL := FALSE;
		VAR_PageSwitch : BOOL := TRUE;
		VAR_ProgressiveId : UINT;
		VAR_BitArray : ARRAY[0..7] OF BOOL;
		VAR_BitIndex : USINT;
		VAR_OldPage : USINT;
		zzEdge00000 : BOOL;
		zzEdge00001 : BOOL;
		zzEdge00002 : BOOL;
		zzEdge00003 : BOOL;
	END_VAR
END_FUNCTION_BLOCK

FUNCTION_BLOCK FB_HMI_ITC_DigitalUsint
	VAR_INPUT
		IN_Visibility : BOOL;
		IN_ReadOnly : BOOL;
		IN_Wait : BOOL;
		IN_Alarm : BOOL;
		IN_IOType : BOOL; (*0: INPUT 1: OUTPUT*)
		IN_Description : STRING[100];
		IN_HMIAutoForce : BOOL;
		IN_BitNumber : INT;
	END_VAR
	VAR_OUTPUT
		OUT_Man : BOOL;
		OUT_ManValue : BOOL;
	END_VAR
	VAR_IN_OUT
		ITC_IO : USINT;
		ITC : BOOL;
		HMI_Data : HMI_ITC_Data_Type;
		HMI_Page : HMI_ITC_Page_Type;
		Index : UINT;
	END_VAR
	VAR
		VAR_Auto : BOOL := TRUE;
		VAR_Man : BOOL := FALSE;
		VAR_PageSwitch : BOOL := TRUE;
		VAR_ProgressiveId : UINT;
		VAR_BitArray : ARRAY[0..7] OF BOOL;
		VAR_BitIndex : USINT;
		VAR_OldPage : USINT;
		zzEdge00000 : BOOL;
		zzEdge00001 : BOOL;
		zzEdge00002 : BOOL;
		zzEdge00003 : BOOL;
	END_VAR
END_FUNCTION_BLOCK

FUNCTION_BLOCK FB_HMI_ITC_DigitalInt
	VAR_INPUT
		IN_Visibility : BOOL;
		IN_ReadOnly : BOOL;
		IN_Wait : BOOL;
		IN_Alarm : BOOL;
		IN_IOType : BOOL; (*0: INPUT 1: OUTPUT*)
		IN_Description : STRING[100];
		IN_HMIAutoForce : BOOL;
		IN_BitNumber : INT;
	END_VAR
	VAR_OUTPUT
		OUT_Man : BOOL;
		OUT_ManValue : BOOL;
	END_VAR
	VAR_IN_OUT
		ITC_IO : INT;
		ITC : BOOL;
		HMI_Data : HMI_ITC_Data_Type;
		HMI_Page : HMI_ITC_Page_Type;
		Index : UINT;
	END_VAR
	VAR
		VAR_Auto : BOOL := TRUE;
		VAR_Man : BOOL := FALSE;
		VAR_PageSwitch : BOOL := TRUE;
		VAR_ProgressiveId : UINT;
		VAR_BitArray : ARRAY[0..15] OF BOOL;
		VAR_BitIndex : USINT;
		VAR_OldPage : USINT;
		zzEdge00000 : BOOL;
		zzEdge00001 : BOOL;
		zzEdge00002 : BOOL;
		zzEdge00003 : BOOL;
	END_VAR
END_FUNCTION_BLOCK

FUNCTION_BLOCK FB_HMI_ITC_AnalogByte
	VAR_INPUT
		IN_Visibility : BOOL;
		IN_ReadOnly : BOOL;
		IN_Wait : BOOL;
		IN_IOType : BOOL; (*0: INPUT 1: OUTPUT*)
		IN_Description : STRING[100];
		IN_MinValue : REAL;
		IN_MaxValue : REAL;
		IN_Unit : STRING[10];
		IN_HMIAutoForce : BOOL;
	END_VAR
	VAR_OUTPUT
		OUT_Man : BOOL;
		OUT_ManValue : BYTE;
	END_VAR
	VAR_IN_OUT
		ITC_IO : BYTE;
		ITC : BYTE;
		HMI_Data : HMI_ITC_Data_Type;
		HMI_Page : HMI_ITC_Page_Type;
		Index : UINT;
	END_VAR
	VAR
		VAR_Man : BOOL := FALSE;
		VAR_ManValue : BYTE := 0;
		VAR_PageSwitch : BOOL := TRUE;
		VAR_ProgressiveId : UINT;
		VAR_OldPage : USINT;
	END_VAR
END_FUNCTION_BLOCK

FUNCTION_BLOCK FB_HMI_ITC_AnalogUsint
	VAR_INPUT
		IN_Visibility : BOOL;
		IN_ReadOnly : BOOL;
		IN_Wait : BOOL;
		IN_IOType : BOOL; (*0: INPUT 1: OUTPUT*)
		IN_Description : STRING[100];
		IN_MinValue : REAL;
		IN_MaxValue : REAL;
		IN_Unit : STRING[10];
		IN_HMIAutoForce : BOOL;
	END_VAR
	VAR_OUTPUT
		OUT_Man : BOOL;
		OUT_ManValue : USINT;
	END_VAR
	VAR_IN_OUT
		ITC_IO : USINT;
		ITC : USINT;
		HMI_Data : HMI_ITC_Data_Type;
		HMI_Page : HMI_ITC_Page_Type;
		Index : UINT;
	END_VAR
	VAR
		VAR_Man : BOOL := FALSE;
		VAR_ManValue : USINT := 0;
		VAR_PageSwitch : BOOL := TRUE;
		VAR_ProgressiveId : UINT;
		VAR_OldPage : USINT;
	END_VAR
END_FUNCTION_BLOCK

FUNCTION_BLOCK FB_HMI_ITC_AnalogInt
	VAR_INPUT
		IN_Visibility : BOOL;
		IN_ReadOnly : BOOL;
		IN_Wait : BOOL;
		IN_IOType : BOOL; (*0: INPUT 1: OUTPUT*)
		IN_Description : STRING[100];
		IN_MinValue : REAL;
		IN_MaxValue : REAL;
		IN_Unit : STRING[10];
		IN_HMIAutoForce : BOOL;
	END_VAR
	VAR_OUTPUT
		OUT_Man : BOOL;
		OUT_ManValue : INT;
	END_VAR
	VAR_IN_OUT
		ITC_IO : INT;
		ITC : INT;
		HMI_Data : HMI_ITC_Data_Type;
		HMI_Page : HMI_ITC_Page_Type;
		Index : UINT;
	END_VAR
	VAR
		VAR_Man : BOOL := FALSE;
		VAR_Value : INT;
		VAR_ManValue : INT := 0;
		VAR_PageSwitch : BOOL := TRUE;
		VAR_ProgressiveId : UINT;
		VAR_OldPage : USINT;
	END_VAR
END_FUNCTION_BLOCK

FUNCTION_BLOCK FB_HMI_ITC_AnalogIntOverUsint
	VAR_INPUT
		IN_Visibility : BOOL;
		IN_ReadOnly : BOOL;
		IN_Wait : BOOL;
		IN_IOType : BOOL; (*0: INPUT 1: OUTPUT*)
		IN_Description : STRING[100];
		IN_MinValue : REAL;
		IN_MaxValue : REAL;
		IN_Unit : STRING[10];
		IN_HMIAutoForce : BOOL;
	END_VAR
	VAR_OUTPUT
		OUT_Man : BOOL;
		OUT_ManValue : INT;
	END_VAR
	VAR_IN_OUT
		ITC_IO : USINT;
		ITC : INT;
		HMI_Data : HMI_ITC_Data_Type;
		HMI_Page : HMI_ITC_Page_Type;
		Index : UINT;
	END_VAR
	VAR
		VAR_Man : BOOL := FALSE;
		VAR_RawValue : INT;
		VAR_Value : INT;
		VAR_ManValue : INT := 0;
		VAR_PageSwitch : BOOL := TRUE;
		VAR_ProgressiveId : UINT;
		VAR_OldPage : USINT;
	END_VAR
END_FUNCTION_BLOCK

FUNCTION_BLOCK FB_HMI_ITC_AnalogUintOverUsint
	VAR_INPUT
		IN_Visibility : BOOL;
		IN_ReadOnly : BOOL;
		IN_Wait : BOOL;
		IN_IOType : BOOL; (*0: INPUT 1: OUTPUT*)
		IN_Description : STRING[100];
		IN_MinValue : REAL;
		IN_MaxValue : REAL;
		IN_Unit : STRING[10];
		IN_HMIAutoForce : BOOL;
	END_VAR
	VAR_OUTPUT
		OUT_Man : BOOL;
		OUT_ManValue : UINT;
	END_VAR
	VAR_IN_OUT
		ITC_IO : USINT;
		ITC : UINT;
		HMI_Data : HMI_ITC_Data_Type;
		HMI_Page : HMI_ITC_Page_Type;
		Index : UINT;
	END_VAR
	VAR
		VAR_Man : BOOL := FALSE;
		VAR_RawValue : UINT;
		VAR_Value : UINT;
		VAR_ManValue : UINT := 0;
		VAR_PageSwitch : BOOL := TRUE;
		VAR_ProgressiveId : UINT;
		VAR_OldPage : USINT;
	END_VAR
END_FUNCTION_BLOCK

FUNCTION_BLOCK FB_HMI_ITC_AnalogDInt
	VAR_INPUT
		IN_Visibility : BOOL;
		IN_ReadOnly : BOOL;
		IN_Wait : BOOL;
		IN_IOType : BOOL; (*0: INPUT 1: OUTPUT*)
		IN_Description : STRING[100];
		IN_MinValue : REAL;
		IN_MaxValue : REAL;
		IN_Unit : STRING[10];
		IN_HMIAutoForce : BOOL;
	END_VAR
	VAR_OUTPUT
		OUT_Man : BOOL;
		OUT_ManValue : DINT;
	END_VAR
	VAR_IN_OUT
		ITC_IO : DINT;
		ITC : DINT;
		HMI_Data : HMI_ITC_Data_Type;
		HMI_Page : HMI_ITC_Page_Type;
		Index : UINT;
	END_VAR
	VAR
		VAR_Man : BOOL := FALSE;
		VAR_Value : DINT;
		VAR_ManValue : DINT := 0;
		VAR_PageSwitch : BOOL := TRUE;
		VAR_ProgressiveId : UINT;
		VAR_OldPage : USINT;
	END_VAR
END_FUNCTION_BLOCK

FUNCTION_BLOCK FB_HMI_ITC_AnalogUdint
	VAR_INPUT
		IN_Visibility : BOOL;
		IN_ReadOnly : BOOL;
		IN_Wait : BOOL;
		IN_IOType : BOOL; (*0: INPUT 1: OUTPUT*)
		IN_Description : STRING[100];
		IN_MinValue : REAL;
		IN_MaxValue : REAL;
		IN_Unit : STRING[10];
		IN_HMIAutoForce : BOOL;
	END_VAR
	VAR_OUTPUT
		OUT_Man : BOOL;
		OUT_ManValue : UDINT;
	END_VAR
	VAR_IN_OUT
		ITC_IO : UDINT;
		ITC : UDINT;
		HMI_Data : HMI_ITC_Data_Type;
		HMI_Page : HMI_ITC_Page_Type;
		Index : UINT;
	END_VAR
	VAR
		VAR_Man : BOOL := FALSE;
		VAR_Value : UDINT;
		VAR_ManValue : UDINT := 0;
		VAR_PageSwitch : BOOL := TRUE;
		VAR_ProgressiveId : UINT;
		VAR_OldPage : USINT;
	END_VAR
END_FUNCTION_BLOCK

FUNCTION_BLOCK FB_HMI_ITC_AnalogDIntOverUsint
	VAR_INPUT
		IN_Visibility : BOOL;
		IN_ReadOnly : BOOL;
		IN_Wait : BOOL;
		IN_IOType : BOOL; (*0: INPUT 1: OUTPUT*)
		IN_Description : STRING[100];
		IN_MinValue : REAL;
		IN_MaxValue : REAL;
		IN_Unit : STRING[10];
		IN_HMIAutoForce : BOOL;
	END_VAR
	VAR_OUTPUT
		OUT_Man : BOOL;
		OUT_ManValue : DINT;
	END_VAR
	VAR_IN_OUT
		ITC_IO : USINT;
		ITC : DINT;
		HMI_Data : HMI_ITC_Data_Type;
		HMI_Page : HMI_ITC_Page_Type;
		Index : UINT;
	END_VAR
	VAR
		VAR_Man : BOOL := FALSE;
		VAR_RawValue : DINT;
		VAR_Value : DINT;
		VAR_ManValue : DINT := 0;
		VAR_PageSwitch : BOOL := TRUE;
		VAR_ProgressiveId : UINT;
		VAR_OldPage : USINT;
	END_VAR
END_FUNCTION_BLOCK

FUNCTION_BLOCK FB_HMI_ITC_AnalogReal
	VAR_INPUT
		IN_Visibility : BOOL;
		IN_ReadOnly : BOOL;
		IN_Wait : BOOL;
		IN_IOType : BOOL; (*0: INPUT 1: OUTPUT*)
		IN_MinValue : REAL;
		IN_MaxValue : REAL;
		IN_Unit : STRING[10];
		IN_Description : STRING[100];
		IN_HMIAutoForce : BOOL;
	END_VAR
	VAR_OUTPUT
		OUT_Man : BOOL;
		OUT_ManValue : REAL;
	END_VAR
	VAR_IN_OUT
		ITC_IO : REAL;
		ITC : REAL;
		HMI_Data : HMI_ITC_Data_Type;
		HMI_Page : HMI_ITC_Page_Type;
		Index : UINT;
	END_VAR
	VAR
		VAR_Man : BOOL := FALSE;
		VAR_Value : REAL;
		VAR_ManValue : REAL := 0.0;
		VAR_PageSwitch : BOOL := TRUE;
		VAR_ProgressiveId : UINT;
		VAR_OldPage : USINT;
	END_VAR
END_FUNCTION_BLOCK

FUNCTION_BLOCK FB_HMI_ITC_AnalogRealOverUsint
	VAR_INPUT
		IN_Visibility : BOOL;
		IN_ReadOnly : BOOL;
		IN_Wait : BOOL;
		IN_IOType : BOOL; (*0: INPUT 1: OUTPUT*)
		IN_MinValue : REAL;
		IN_MaxValue : REAL;
		IN_Unit : STRING[10];
		IN_Description : STRING[100];
		IN_HMIAutoForce : BOOL;
	END_VAR
	VAR_OUTPUT
		OUT_Man : BOOL;
		OUT_ManValue : REAL;
	END_VAR
	VAR_IN_OUT
		ITC_IO : USINT;
		ITC : REAL;
		HMI_Data : HMI_ITC_Data_Type;
		HMI_Page : HMI_ITC_Page_Type;
		Index : UINT;
	END_VAR
	VAR
		VAR_Man : BOOL := FALSE;
		VAR_RawValue : REAL;
		VAR_Value : REAL;
		VAR_ManValue : REAL := 0.0;
		VAR_PageSwitch : BOOL := TRUE;
		VAR_ProgressiveId : UINT;
		VAR_OldPage : USINT;
		RealValue : REAL;
	END_VAR
END_FUNCTION_BLOCK

FUNCTION_BLOCK FB_HMI_ITC_End
	VAR_INPUT
		IN_IODigAnalog : BOOL; (*0: DIGITAL 1: ANALOG*)
		IN_IOType : BOOL; (*0: INPUT 1: OUTPUT*)
	END_VAR
	VAR_IN_OUT
		HMI_Data : HMI_ITC_Data_Type;
		HMI_Page : HMI_ITC_Page_Type;
		Index : UINT;
	END_VAR
	VAR
		VAR_ProgressiveId : UINT;
		i : UINT;
	END_VAR
END_FUNCTION_BLOCK

FUNCTION_BLOCK FB_HMI_ITC_FastDigitalByte
	VAR_INPUT
		IN_Visibility : BOOL;
		IN_ReadOnly : BOOL;
		IN_Wait : BOOL;
		IN_Alarm : BOOL;
		IN_IOType : BOOL; (*0: INPUT 1: OUTPUT*)
		IN_Description : STRING[100];
		IN_HMIAutoForce : BOOL;
		ITC : BOOL;
	END_VAR
	VAR_OUTPUT
		OUT_Man : BOOL;
		OUT_ManValue : BOOL;
	END_VAR
	VAR_IN_OUT
		HMI_Data : HMI_ITC_Data_Type;
		HMI_Page : HMI_ITC_Page_Type;
		Index : UINT;
	END_VAR
	VAR
		VAR_Auto : BOOL := TRUE;
		VAR_Man : BOOL := FALSE;
		VAR_PageSwitch : BOOL := TRUE;
		VAR_ProgressiveId : UINT;
		VAR_OldPage : USINT;
		zzEdge00000 : BOOL;
		zzEdge00001 : BOOL;
		zzEdge00002 : BOOL;
		zzEdge00003 : BOOL;
	END_VAR
END_FUNCTION_BLOCK

FUNCTION_BLOCK FB_HMI_ITC_FastAnalogInt
	VAR_INPUT
		IN_Visibility : BOOL;
		IN_ReadOnly : BOOL;
		IN_Wait : BOOL;
		IN_IOType : BOOL; (*0: INPUT 1: OUTPUT*)
		IN_Description : STRING[100];
		IN_MinValue : REAL;
		IN_MaxValue : REAL;
		IN_Unit : STRING[10];
		IN_HMIAutoForce : BOOL;
		ITC : INT;
	END_VAR
	VAR_OUTPUT
		OUT_Man : BOOL;
		OUT_ManValue : INT;
	END_VAR
	VAR_IN_OUT
		HMI_Data : HMI_ITC_Data_Type;
		HMI_Page : HMI_ITC_Page_Type;
		Index : UINT;
	END_VAR
	VAR
		VAR_Man : BOOL := FALSE;
		VAR_ManValue : INT := 0;
		VAR_PageSwitch : BOOL := TRUE;
		VAR_ProgressiveId : UINT;
		VAR_OldPage : USINT;
	END_VAR
END_FUNCTION_BLOCK

FUNCTION_BLOCK FB_HMI_ITC_FastAnalogDInt
	VAR_INPUT
		IN_Visibility : BOOL;
		IN_ReadOnly : BOOL;
		IN_Wait : BOOL;
		IN_IOType : BOOL; (*0: INPUT 1: OUTPUT*)
		IN_Description : STRING[100];
		IN_MinValue : REAL;
		IN_MaxValue : REAL;
		IN_Unit : STRING[10];
		IN_HMIAutoForce : BOOL;
		ITC : DINT;
	END_VAR
	VAR_OUTPUT
		OUT_Man : BOOL;
		OUT_ManValue : DINT;
	END_VAR
	VAR_IN_OUT
		HMI_Data : HMI_ITC_Data_Type;
		HMI_Page : HMI_ITC_Page_Type;
		Index : UINT;
	END_VAR
	VAR
		VAR_Man : BOOL := FALSE;
		VAR_ManValue : DINT := 0;
		VAR_PageSwitch : BOOL := TRUE;
		VAR_ProgressiveId : UINT;
		VAR_OldPage : USINT;
	END_VAR
END_FUNCTION_BLOCK

FUNCTION_BLOCK FB_Counter
	VAR_INPUT
		IN_Clock1Hz : BOOL;
		IN_TimeCondition : BOOL;
		IN_IncrementCondition : BOOL;
		IN_PulseWeight : REAL;
		IN_Reset : BOOL;
		IN_Date : DATE_AND_TIME;
	END_VAR
	VAR_IN_OUT
		IN_OUT_CounterPartialStruct : Counters_Type;
		IN_OUT_CounterTotalStruct : Counters_Type;
	END_VAR
	VAR
		tempReal : REAL := 0.0;
	END_VAR
END_FUNCTION_BLOCK

FUNCTION FC_Counter : BOOL (* *) (*$GROUP=User,$CAT=User,$GROUPICON=User.png,$CATICON=User.png*)
	VAR_INPUT
		IN_Clock1Hz : BOOL;
		IN_TimeCondition : BOOL;
		IN_IncrementCondition : BOOL;
		IN_Reset : BOOL;
		IN_Date : DATE_AND_TIME;
	END_VAR
	VAR_IN_OUT
		IN_OUT_CounterPartialStruct : Counters_Type;
		IN_OUT_CounterTotalStruct : Counters_Type;
	END_VAR
END_FUNCTION

FUNCTION FC_IncTimer : BOOL (* *) (*$GROUP=User,$CAT=User,$GROUPICON=User.png,$CATICON=User.png*)
	VAR_INPUT
		IN_Clock1Hz : BOOL;
		IN_Condition : BOOL;
		IN_Reset : BOOL;
	END_VAR
	VAR_IN_OUT
		IN_OUT_CounterStruct : CounterTime_Type;
	END_VAR
END_FUNCTION

FUNCTION FC_SpeedCheck : BOOL (* *) (*$GROUP=User,$CAT=User,$GROUPICON=User.png,$CATICON=User.png*)
	VAR_INPUT
		IN_SpeedReq : REAL;
		IN_SpeedAct : REAL;
		IN_Mode : USINT; (*0 = Equal
1 = Greater
2 = Lower*)
	END_VAR
END_FUNCTION

FUNCTION FC_ReminderShift : INT (*Reminder With Minimum Value*) (*$GROUP=User,$CAT=User,$GROUPICON=User.png,$CATICON=User.png*)
	VAR_INPUT
		Dividend : INT;
		Divisor : INT;
		Start : INT;
	END_VAR
	VAR
		ReminderA : INT;
		ReminderB : INT;
		ReminderC : INT;
		LocalDivisor : INT;
	END_VAR
END_FUNCTION

FUNCTION FC_MacaoTimer : BOOL (* *) (*$GROUP=User,$CAT=User,$GROUPICON=User.png,$CATICON=User.png*)
	VAR_INPUT
		IN_Clock1Hz : BOOL;
		IN_Condition : BOOL;
		IN_Reset : BOOL;
	END_VAR
	VAR_IN_OUT
		IN_OUT_Counter : UDINT;
	END_VAR
END_FUNCTION

FUNCTION_BLOCK Integral
	VAR_INPUT
		IN_NewValue : REAL; (*New value*)
		IN_IntCycle : REAL; (*Cycle time*)
	END_VAR
	VAR_IN_OUT
		OUT_Integral : REAL; (*Integrated value*)
	END_VAR
	VAR
		VAR_OldValue : REAL := 0.0; (*Old value*)
	END_VAR
END_FUNCTION_BLOCK

FUNCTION_BLOCK LevelVariation
	VAR_INPUT
		IN_Enable : BOOL; (*Function Enable*)
		IN_TankVolumePV : REAL; (*Actual Tank Volume [l]*)
		IN_ControlTime : REAL; (*Level Control Scan Time  [s]*)
	END_VAR
	VAR_OUTPUT
		OUT_Low : BOOL; (*Low Flow Required*)
		OUT_High : BOOL; (*High Flow Required*)
	END_VAR
	VAR
		OldVolume : REAL;
		VAR_RTInfo : RTInfo;
		Timer : REAL;
		VAR_Cycle : REAL;
		DeltaVolume : REAL;
		AbsoluteError : REAL; (*Level Error (no sign)*)
		RestoreTime : REAL; (*Number of Cycles with no Negative Variation*)
	END_VAR
	VAR CONSTANT
		RestoreTimeLimit : REAL := 50.0; (*Number of Cycles Limit with no Negative Variation*)
	END_VAR
	VAR
		RestoreError : REAL; (*Number of Cycles in Idle*)
	END_VAR
	VAR CONSTANT
		RestoreErrorLimit : REAL := 50.0; (*Number of Cycles Limit in Idle*)
	END_VAR
END_FUNCTION_BLOCK

FUNCTION_BLOCK PID_Cont
	VAR_INPUT
		IN_ConfigPresent : BOOL; (*Enables PID execution and visualization on HMI*)
		IN_ConfigEngValue : BOOL; (*Configuration: FF and PID OUT Scale - TRUE-> 0-100%, FALSE-> Ing.Unit.*)
		IN_Reverse : BOOL; (*Reverse action (bigger the error smaller the output)*)
		IN_Gain : REAL; (*Proportional gain*)
		IN_TI : REAL; (*Reset time*)
		IN_TD : REAL; (*Derivative time*)
		IN_PV : REAL; (*Process Value for PID Control*)
		IN_Auto : BOOL; (*Execute PID calculations*)
		IN_FixOut : BOOL;
		IN_FixOutValue : REAL;
		IN_IntHold : BOOL; (*Integral action hold*)
		IN_AutoSP : REAL; (*Set Point for PID Control*)
		IN_Disv : REAL; (*Disturbance variable (same unit as manipulated value)*)
		IN_MaxScale : REAL; (*Maximum scale value*)
		IN_Slew : BOOL; (*Slew on SP required*)
		IN_SPSlew : REAL; (*Set Point slew*)
		IN_MinDev : REAL; (*To Set Point Low Deviation (for SP obtained)*)
		IN_MaxDev : REAL; (*To Set Point High Deviation (for SP obtained)*)
		IN_OutMin : REAL; (*Output minimum value*)
		IN_OutMax : REAL; (*Output maximum value*)
		IN_CycleTime : TIME;
		IN_TIInit : BOOL;
		IN_TIInitValue : REAL;
	END_VAR
	VAR_OUTPUT
		OUT : REAL; (*Manipulated value*)
		OUT_ActSP : REAL;
		OUT_Error : REAL; (*Error signal [eng]*)
		OUT_P : REAL; (*Proportionality component*)
		OUT_I : REAL; (*Integral component*)
		OUT_D : REAL; (*Derivative component*)
	END_VAR
	VAR_IN_OUT
		HMI : HMI_PID_Type;
	END_VAR
	VAR
		LCRLimScal_PV : LCRLimScal;
		LCRLimScal_SP : LCRLimScal;
		VAR_Derivative : REAL;
		VAR_FirstCycle : BOOL;
		VAR_GainError : REAL;
		VAR_Integral : Integral;
		VAR_IntegralBlock : BOOL; (*Freeze Integral Calculation*)
		VAR_IntegralOut : REAL;
		VAR_IntegralSaturation : BOOL;
		LCRRamp : LCRRamp;
		VAR_OldError : REAL;
		VAR_Proportional : REAL;
		VAR_RTInfo : RTInfo;
		VAR_SPRamped : REAL;
		VAR_SP : REAL;
		VAR_PV : REAL;
		VAR_CycleCounter : REAL;
		VAR_CycleTime : REAL;
		VAR_SlewInit : BOOL;
		TON_Cycle : TON;
		zzEdge00000 : BOOL;
		zzEdge00001 : BOOL;
		zzEdge00002 : BOOL;
	END_VAR
END_FUNCTION_BLOCK

FUNCTION_BLOCK PID_FF_Mod
	VAR_INPUT
		IN_Enable : BOOL; (*Feed Forward Enable (Bit true)*)
		IN_Reset : BOOL; (*Feed Forward Reset (Bit true)*)
		IN_Raise_Step : REAL; (*Raise Ramp Step Start Delay (0 -:- 100)*)
		IN_Raise_Step_Counter : REAL; (*Raise Ramp Step Start Delay Counter*)
		IN_Lower_Step : REAL; (*Lower  Ramp Step Start Delay (0 -:- 100)*)
		IN_Lower_Step_Counter : REAL; (*Lower Ramp Step Start Delay Counter*)
		IN_FF_SP1 : REAL; (*Feed Forward Set Point 1 Value (High Set Point)*)
		IN_FF_SP2 : REAL; (*Feed Forward Set Point 2 Value (High Set Point)*)
		IN_SP1_SP2_Time : REAL; (*Time delay before Lower Ramp to Feed Forward Set Point 2*)
		IN_Ramp_Speed : REAL; (*Feed Forward Ramp Speed (Raise-Lower)*)
		IN_Actual_Speed : REAL; (*Actual Machine Speed (c/h)*)
		IN_Size_Speed : REAL; (*Max Machine Speed for actual Container Size (c/h)*)
	END_VAR
	VAR_OUTPUT
		OUT_FF_Value : REAL;
		OUT_FF_Value_Int : INT;
	END_VAR
	VAR
		Running : BOOL;
		Lower_Ramp : BOOL;
		SP1_ON : BOOL;
		SP2_ON : BOOL;
		FF_SP1_Recipe : REAL;
		Speed : REAL;
		Max_Speed : REAL;
		FF_SP1_Val : REAL;
		Ramp_Time : REAL;
		Ramp_Speed_R : REAL;
		Ramp_Value : REAL;
		FF_value_Out : REAL;
		FF_SP2_Save : REAL;
		FF_SP2_Time : TON;
		FF_SP2_Recipe : REAL;
		FF_SP2_Val : REAL;
	END_VAR
END_FUNCTION_BLOCK

FUNCTION_BLOCK PID_FF_Pump
	VAR_INPUT
		IN_Enable : BOOL; (*Feed Forward Enable (Bit true)*)
		IN_Reset : BOOL;
		IN_Control_Type : BOOL; (*0=Control on Ring;1=Control on Product Pipe*)
		IN_FV_Number : REAL; (*Filling Valves Number*)
		IN_RingDiameter_mm : REAL;
		IN_FV_FromFloor : REAL; (*Water From The Floor on The Product Level Tank [mm]*)
		IN_PTF_FromFloor : REAL; (*Water From The Floor on The Product Level Tank [mm]*)
		IN_PTF_FromFV : REAL; (*Water From The Floor on The Product Level Tank [mm]*)
		IN_Pump_Kf : REAL;
		IN_Pump_Kpc : REAL;
		IN_Pump_OutMax : REAL;
		IN_FMCActualFlowrate : REAL;
		IN_TankLevel_mm : REAL; (*Water From The Floor on The Product Level Tank [mm]*)
		IN_Actual_SPmm : REAL; (*Actual Machine Speed (B/h)*)
		IN_Actual_PVmm : REAL; (*Actual Machine Speed (B/h)*)
		IN_Actual_SPbar : REAL; (*Actual Machine Speed (B/h)*)
		IN_Actual_PVbar : REAL; (*Actual Machine Speed (B/h)*)
		IN_Actual_Speed : REAL; (*Actual Machine Speed (B/h)*)
	END_VAR
	VAR_OUTPUT
		OUT_FF : REAL;
		OUT_PID_PV : REAL;
		OUT_PID_SP : REAL;
		OUT_Error : BOOL;
	END_VAR
	VAR
		Radius : REAL;
		Omega : REAL;
		CentrifugalForce : REAL;
		Level_SP_Calculated : REAL;
		Pid_PV_Calculated : REAL;
		PV_Product_Pump : REAL;
		Kpc_FlowRate_Filling : REAL;
		Real_Level : REAL;
	END_VAR
END_FUNCTION_BLOCK

FUNCTION_BLOCK PID_FF_PumpH
	VAR_INPUT
		IN_Enable : BOOL; (*Feed Forward Enable (Bit true)*)
		IN_Reset : BOOL;
		IN_Control_Type : BOOL; (*0=Control on Ring;1=Control on Product Pipe*)
		IN_FV_Number : REAL; (*Filling Valves Number*)
		IN_RingDiameter_mm : REAL;
		IN_FV_FromFloor : REAL; (*Water From The Floor on The Product Level Tank [mm]*)
		IN_PTF_FromFloor : REAL; (*Water From The Floor on The Product Level Tank [mm]*)
		IN_PTF_FromFV : REAL; (*Water From The Floor on The Product Level Tank [mm]*)
		IN_Pump_Kf : REAL;
		IN_Pump_Kpc : REAL;
		IN_Pump_OutMax : REAL;
		IN_PumpMaxFillingTime : REAL;
		IN_FMCActualFlowrate : REAL;
		IN_FMCAverFillingTime : REAL;
		IN_FMCStepStartFilling : REAL;
		IN_FMCStepExitCam : REAL;
		IN_TankLevel_mm : REAL; (*Water From The Floor on The Product Level Tank [mm]*)
		IN_Actual_SPmm : REAL; (*Actual Machine Speed (c/h)*)
		IN_Actual_PVmm : REAL; (*Actual Machine Speed (c/h)*)
		IN_Actual_SPbar : REAL; (*Actual Machine Speed (c/h)*)
		IN_Actual_PVbar : REAL; (*Actual Machine Speed (c/h)*)
		IN_Actual_Speed : REAL; (*Actual Machine Speed (c/h)*)
		IN_Recipe_Speed : REAL; (*Max Machine Speed for actual Container Size (c/h)*)
	END_VAR
	VAR_OUTPUT
		OUT_FF : REAL;
		OUT_Centifrugal : REAL;
		OUT_Error : BOOL;
	END_VAR
	VAR
		Radius : REAL;
		Omega : REAL;
		CentrifugalForce : REAL;
		MAX_FillingTime : REAL;
		MAX_ContainersNumber : REAL;
		Level_SP_Calculated : REAL;
		FillingTime : REAL;
		Calculated_FillingTime : REAL;
		PV_Product_Pump : REAL;
		Kpc_FlowRate_Filling : REAL;
		Real_Level : REAL;
	END_VAR
END_FUNCTION_BLOCK

FUNCTION_BLOCK RCP_Management
	VAR_INPUT
		IN_AdrPLCRecipe : {REDUND_UNREPLICABLE} UDINT; (*Temporary structure from HMI*)
		IN_AdrHMIRecipe : {REDUND_UNREPLICABLE} UDINT; (*PLC Internal Structure*)
		IN_SizePLCRecipe : UDINT;
		IN_SizeHMIRecipe : UDINT;
		IN_RequestedRCP : STRING[150];
		IN_DownloadRequest : BOOL;
	END_VAR
	VAR_OUTPUT
		OUT_ParameterError : BOOL;
		OUT_RecipeLoaded : BOOL;
		OUT_Step : RCP_Management_Step;
	END_VAR
	VAR_IN_OUT
		RCP_Manag : RCP_Management_Type;
	END_VAR
	VAR
		VAR_FirstCycle : BOOL;
		VAR_Step_old : RCP_Management_Step;
		TMR_tonRCP_WaitRestart : TON;
		TMR_tonRCP_WaitStart : TON;
		TMR_tonRCP_DownloadTimeOut : TON;
	END_VAR
END_FUNCTION_BLOCK

FUNCTION_BLOCK Sequencer_v1
	VAR_INPUT
		IN_StepConfig : SEQ_StepConfig_Type;
		IN_T_TimeClock : BOOL;
		IN_Step : UINT;
		IN_StepCounter : UINT;
		IN_Pause_Request : BOOL;
		IN_FillingValveNr : UINT;
	END_VAR
	VAR_OUTPUT
		OUT_TON_Time_END : BOOL;
		OUT_TO_Time_END : BOOL;
		OUT_T_Time_END : BOOL;
		OUT_LapsCounterRequest : BOOL;
		OUT_Laps_Done : BOOL;
		OUT_Cycles_Done : BOOL;
		OUT_HMI_ID : UINT; (*ID to match text on HMI*)
		OUT_JMP_StepPrevious : UINT; (*Step wich the sequence is coming from*)
		OUT_JMP_Step : UINT;
		OUT_Laps_Progress : UINT; (*Progress of Laps Executed*)
		OUT_StepTimePr_TON : UINT; (*TON Preset Time*)
		OUT_StepTimePr_T : UINT; (*T Preset Time*)
		OUT_StepTimeCV_TON : UINT; (*TON ActualTime*)
		OUT_StepTimeCV_T : UINT; (*T Actual Time*)
	END_VAR
	VAR_IN_OUT
		CyclesCounter : UDINT;
	END_VAR
	VAR
		TON_Time : TON;
		TO_Time : TON;
		T_Time : CTU;
		VAR_ChangeInProgress : BOOL;
		VAR_CounterInitialized : BOOL;
	END_VAR
END_FUNCTION_BLOCK

FUNCTION_BLOCK Sequencer_v2
	VAR_INPUT
		IN_StepConfig : SEQ_StepConfig_Type;
		IN_T_TimeClock : BOOL;
		IN_Step : UINT;
		IN_StepCounter : UINT;
		IN_Pause_Request : BOOL;
		IN_FillingValveNr : UINT;
	END_VAR
	VAR_OUTPUT
		OUT_TON_Time_END : BOOL;
		OUT_TO_Time_END : BOOL;
		OUT_T_Time_END : BOOL;
		OUT_LapsCounterRequest : BOOL;
		OUT_Laps_Done : BOOL;
		OUT_Cycles_Done : BOOL;
		OUT_HMI_ID : UINT; (*ID to match text on HMI*)
		OUT_StepPrevious : UINT; (*Step wich the sequence is coming from*)
		OUT_StepActual : UINT;
		OUT_Laps_Progress : UINT; (*Progress of Laps Executed*)
		OUT_StepTimePr_TON : UINT; (*TON Preset Time*)
		OUT_StepTimePr_T : UINT; (*T Preset Time*)
		OUT_StepTimeCV_TON : UINT; (*TON ActualTime*)
		OUT_StepTimeCV_T : UINT; (*T Actual Time*)
		OUT_StepProgressiveTime : UINT; (*T Actual Time*)
	END_VAR
	VAR_IN_OUT
		CyclesCounter : UDINT;
	END_VAR
	VAR
		TON_Time : TON;
		TO_Time : TON;
		T_StepProgressiveTime : TON;
		T_Time : CTU;
		VAR_ChangeInProgress : BOOL;
		VAR_CounterInitialized : BOOL;
	END_VAR
END_FUNCTION_BLOCK

FUNCTION_BLOCK TankMultiScale
	VAR_INPUT
		IN_ConfigPresent : BOOL;
		IN_Wait : BOOL;
		IN_Sp_Type : USINT; (*[1=Wait percentage SP] [2=Wait Volume SP] [3=Wait level Height]*)
		IN_TNK_PV : REAL;
		IN_TNK_LowLimitAbs : REAL;
		IN_TNK_Diameter_mm : REAL;
		IN_TNK_Bottom_liters : REAL;
		IN_ProbeLength_mm : REAL;
		IN_FromFloor_ToZeroProbe_mm : REAL;
		IN_Scale : ARRAY[0..3] OF IN_Analog_Multiscale; (*0..3 = Arrays for Different Scale*)
	END_VAR
	VAR_OUTPUT
		OUT_Scale : ARRAY[0..3] OF OUT_Analog_Multiscale;
	END_VAR
	VAR_IN_OUT
		HMI : HMI_Analog_Multiscale_Type;
	END_VAR
	VAR
		pi : REAL;
		diameter_cm : REAL;
		r_cm : REAL; (*radius [cm]*)
		heightAck_cm : REAL;
		volumeAck_cm3 : REAL;
		volumeAck_liters : REAL;
		heightTot_cm : REAL;
		volumeTot_cm3 : REAL;
		volumeTot_liters : REAL;
		LowLimitAbs_cm : REAL;
		LowLimitAbs_cm3 : REAL;
		LowLimitAbs_liters : REAL;
	END_VAR
END_FUNCTION_BLOCK

FUNCTION_BLOCK Siko_Management
	VAR_INPUT
		IN_Mode : INT; (*0: Idle ; 1: Production ; 2: Cleaning*)
		IN_HMI_MotEnable : BOOL;
		IN_HMI_ManualEnable : BOOL;
		IN_HMI_StartWrite : BOOL;
		IN_HMI_Calibrate : BOOL;
		IN_HMI_StartRead : BOOL;
		IN_HMI_JogForward : BOOL;
		IN_HMI_JogBackward : BOOL;
		IN_HMI_MoveAt : BOOL;
		IN_PosProduction : REAL;
		IN_PosCleaning : REAL;
		IN_PosManualSP : REAL;
		IN_EnableToRun : BOOL; (*//v049*)
		IN_Reset : BOOL;
	END_VAR
	VAR_OUTPUT
		OUT_Running : BOOL;
		OUT_Done : BOOL;
		OUT_PositionError : BOOL;
	END_VAR
	VAR_IN_OUT
		IN_SikoData : SIKO_MASTER_Type;
	END_VAR
	VAR
		CalculateSP : REAL;
		Status : INT;
		StepTimer : TON;
		zzEdge00000 : BOOL;
		zzEdge00001 : BOOL;
	END_VAR
END_FUNCTION_BLOCK

FUNCTION_BLOCK Siko_FB
	VAR_INPUT
		IN_EmergencyOK : BOOL;
		IN_Reset : BOOL;
		IN_CommunicationOK : BOOL;
		IN_TimeOutPositioning : TIME;
		IN_PGain : REAL;
		IN_IGain : REAL;
		IN_DGain : REAL;
		IN_VPos : REAL;
		IN_APos : REAL;
		IN_VJog : REAL;
		IN_PosWindows : REAL;
		IN_GearIn : REAL;
		IN_GearOut : REAL;
		IN_SpindlePitch : REAL;
		IN_SenseOfRotation : REAL;
		IN_UpperLimit : REAL;
		IN_LowerLimit : REAL;
		IN_CalibrationValue : REAL;
	END_VAR
	VAR_IN_OUT
		DeviceData : SIKO_MASTER_Type;
		IO : SIKO_COM_Type;
	END_VAR
	VAR
		Com : SIKO_COM_Type;
		ReloadData : BOOL;
		KFactorReal : REAL;
		CounterRead : SINT;
		CounterWrite : SINT;
		CounterCalibration : SINT;
		ReadOrWriteInProgress : BOOL;
		TReadAndWrite : TON;
		zzEdge00000 : BOOL;
		SwitchOn : BOOL;
		TPowerOn : TOF;
		PositionFinished : BOOL;
		zzEdge00001 : BOOL;
		RisingFrontRead : BOOL;
		zzEdge00002 : BOOL;
		RisingFrontWrite : BOOL;
		zzEdge00003 : BOOL;
		zzEdge00004 : BOOL;
		Temp_HIW : UDINT;
		Temp_HSW : UDINT;
		Temp_IN_PWE : UDINT;
		Temp_OUT_PWE : UDINT;
	END_VAR
END_FUNCTION_BLOCK

FUNCTION_BLOCK TP_Reset
	VAR_INPUT
		IN : BOOL;
		PT : TIME;
		RESET : BOOL;
	END_VAR
	VAR_OUTPUT
		Q : BOOL;
	END_VAR
	VAR
		TimeCounter : UDINT;
		RT_Info : RTInfo;
		zzEdge00000 : BOOL;
		zzEdge00001 : BOOL;
	END_VAR
END_FUNCTION_BLOCK

FUNCTION_BLOCK FB_VFD_DataRead (*v999Daq*)
	VAR_INPUT
		IN_ReadDataEnable : BOOL;
		IN_DeviceAddress : UDINT;
		IN_DeviceNode : USINT;
		IN_DeviceName : STRING[80];
		IN_DanfossFC280 : BOOL;
		IN_IO_PlkVFD_FC280 : IO_PLK_DanfossFC280_Drive_Type;
		IN_IO_PlkVFD : IO_PLK_Danfoss_Drive_Type;
	END_VAR
	VAR_OUTPUT
		OUT_Error : BOOL;
	END_VAR
	VAR_IN_OUT
		VfdData : Vfd_Data_Type;
	END_VAR
	VAR
		Danfoss_Comm : EplSDORead;
		VAR_DataReadIndex : INT;
		TON_Read : TON;
	END_VAR
END_FUNCTION_BLOCK

FUNCTION_BLOCK FB_Flip
	VAR_INPUT
		IN_CycleOn : BOOL;
		IN_CyclePause : BOOL;
		IN_CycleLoop : BOOL;
		IN_CycleStartOffCount : BOOL;
		IN_CycleNrReset : BOOL;
		IN_CycleNr : UDINT;
		IN_CycleTimeOn : UDINT;
		IN_CycleTimeOff : UDINT;
	END_VAR
	VAR_OUTPUT
		OUT_CycleNr : UDINT;
		OUT_CycleTimeOn : UDINT;
		OUT_CycleTimeOff : UDINT;
		OUT_CycleDone : BOOL;
		Out : BOOL;
	END_VAR
	VAR
		Command_State : USINT;
		VAR_CycleTimeOn : UDINT;
		VAR_CycleTimeOff : UDINT;
		VAR_CycleNr : UDINT;
		VAR_CyleOn : BOOL;
		VAR_CyleCntOn : BOOL;
		VAR_CyleCntOff : BOOL;
		VAR_CyleOnTimeReset : BOOL;
		VAR_CyleOffTimeReset : BOOL;
		VAR_CyleNrReset : BOOL;
		VAR_CycleOffDone : BOOL;
		VAR_CycleOnDone : BOOL;
		VAR_CycleNrDone : BOOL;
		TON_Blink : TON;
		zzEdge00000 : BOOL;
		zzEdge00001 : BOOL;
		zzEdge00002 : BOOL;
	END_VAR
END_FUNCTION_BLOCK
```

#### Types.typ
```iecst
TYPE
	AlarmCmd_Type : 	STRUCT
		ActionEn : BOOL := TRUE; (*If TRUE the action is performed; If FALSE the alarm is shown as a Message*)
		ByPassEn : BOOL;
		ByPass : BOOL;
		ActionDis : BOOL;
		Active : BOOL; (*If TRUE the alarm is activated.*)
		Visibility : BOOL := TRUE; (*If TRUE the HMI show the Alarm. The action will always performed*)
		DependentActive : BOOL; (*If TRUE the Alarm is deactivated by its master alarm V4.A.A.1.6.13*)
	END_STRUCT;
	AlarmCFG_Type : 	STRUCT
		Action : USINT;
		Category : USINT;
		OMAC_Code : UINT;
		OMAC_Index : UINT;
	END_STRUCT;
	ActionSum_Type : 	STRUCT
		Bit : UDINT;
	END_STRUCT;
	ActionSum_Enum :
		( (*V4.A.A.1.6.13*)
		ALR_NULL := 0, (*No Action, No Code*)
		ALR_MS_QuickStop := 1, (*Machine Stop: Fast deceleration ramp*)
		ALR_MS_NormalStop := 2, (*Machine Stop: Low deceleration ramp*)
		ALR_MS_QuickWithJog := 3, (*Machine Stop: Fast deceleration ramp + JOG Running Possible*)
		ALR_MS_NormalWithJog := 4, (*Machine Stop: Low deceleration ramp + JOG Running Possible*)
		ALR_MS_NormalWithJogMnt := 5, (*Machine Stop Auto Reset: Low deceleration ramp + JOG Running Possible*)
		ALR_CSR := 6, (*Container Stop Operator Reset: Immediate*)
		ALR_CSR_AfterSlowdown := 7, (*Container Stop Operator Reset: After Slowing*)
		ALR_CSR_StopAfterEmptying := 8, (*Container Stop Operator Reset: Emptying + Machine Normal Stop*)
		ALR_CSA := 9, (*Container Stop Auto Reset: Immediate*)
		ALR_CSA_AfterSlowdown := 10, (*Container Stop Auto Reset: After Slowing*)
		ALR_StartModeDisabled := 30, (*Start-Up Function Mode Disabled*)
		ALR_NoProduction := 31 (*No Action, Production Suspended (only Data Acquisition Code)*)
		);
	RCP_Management_Type : 	STRUCT
		Enable : BOOL; (*To HMI - Enable to download a recipe*)
		Started : BOOL; (*From HMI - Download Started*)
		Ended : BOOL; (*From HMI - Download Ended*)
		Received : BOOL; (*To HMI - Ended Received *)
		EditOnlineEnable : BOOL; (*To HMI - Edit Online Enabled*)
		EditOnlineActive : BOOL; (*From HMI - Edit Online Active*)
		ActiveRecipeName : STRING[70]; (*From HMI - Name of Actived Recipe*)
		RequestedRecipeName : STRING[70]; (*To HMI - Name of the requested recipe*)
		DownloadRequest : BOOL; (*To HMI - Request command to download a recipe*)
	END_STRUCT;
	RCP_Management_Step :
		(
		Wait_Download := 0,
		Download_Request := 1,
		Copy_To_Internal := 2,
		Download_Done := 3,
		Clear_Cmd := 4,
		Edit_Online := 10,
		Download_Error := 20
		);
	HMI_ITC_Page_Type : 	STRUCT
		PartnerID : USINT := 11;
		PageNum : USINT := 0;
	END_STRUCT;
	HMI_ITC_Data_Type : 	STRUCT
		PartnerID : USINT;
		ComType : USINT;
		ComAddress : STRING[35];
		LocalPort : UINT; (*Local port number used to Receive*)
		RemotePort : UINT; (*Remote port number used o Send*)
		ComSwap : BOOL;
		PageUp : HMI_ITC_PB_Type := (Visibility:=TRUE);
		PageDown : HMI_ITC_PB_Type := (Visibility:=TRUE);
		ComStatus : USINT;
		ComMask : HMI_ITC_SS2P_Type := (Visibility:=TRUE);
		DigitalIn : ARRAY[1..16]OF HMI_DigitalITC_Type;
		AnalogIn : ARRAY[1..4]OF HMI_AnalogITC_Type;
		DigitalOut : ARRAY[1..16]OF HMI_DigitalITC_Type;
		AnalogOut : ARRAY[1..4]OF HMI_AnalogITC_Type;
		ManActive : BOOL;
	END_STRUCT;
	HMI_AnalogITC_Type : 	STRUCT
		Visibility : BOOL;
		PV : REAL;
		Unit : STRING[10];
		Wait : BOOL;
		MinValue : REAL;
		MaxValue : REAL;
		Enable : BOOL;
		Man : BOOL;
		PV_Man : REAL;
		Description : STRING[100];
		Decimal : USINT;
	END_STRUCT;
	HMI_DigitalITC_Type : 	STRUCT
		Visibility : BOOL;
		Enable : BOOL;
		Auto : BOOL := TRUE;
		LampState : BOOL;
		Alarm : BOOL;
		Wait : BOOL;
		Man : BOOL;
		Description : STRING[100];
	END_STRUCT;
	HMI_ITC_PB_Type : 	STRUCT  (*Push button (ON-OFF;) 0=OFF - 1=ON*)
		Enable : BOOL; (*State: Command Enabled*)
		LampON : BOOL; (*State: Lamp Command ON*)
		Blink : BOOL; (*State: Blink LampOn*)
		Visibility : BOOL; (*Configuration: Present*)
		ON : BOOL; (*Command: Push Button ON*)
	END_STRUCT;
	HMI_ITC_SS2P_Type : 	STRUCT  (*Selector 2 position (Auto-Man; ON-OFF;) 0=Auto/OFF - 1=Man/ON*)
		Enable : BOOL; (*State: Command Enabled*)
		LampON : BOOL; (*State: Lamp Command ON*)
		Blink : BOOL; (*State: Blink LampOn*)
		Visibility : BOOL; (*Configuration: Present*)
		ON : BOOL; (*Command: Push Button ON*)
	END_STRUCT;
	IO_TimeClock_Type : 	STRUCT
		Seconds : UDINT;
		Nanoseconds : UDINT;
	END_STRUCT;
	Counters_Type : 	STRUCT
		CounterValue : UDINT;
		CounterTime : CounterTime_Type;
		StartDate : DINT;
	END_STRUCT;
	CounterTime_Type : 	STRUCT
		Day : UINT;
		Hour : USINT;
		Min : USINT;
		Sec : USINT;
	END_STRUCT;
	HMI_ComboBoxElements_Type : 	STRUCT
		Present : BOOL;
		Name : STRING[20];
	END_STRUCT;
	SEQ_StepConfig_Type : 	STRUCT
		T_TimePr : UINT;
		TO_TimePr : UINT;
		HMI_ID : UINT;
		TON_TimePr : UINT;
		Laps_Request : UINT;
		Cycle_Pr : UINT;
		TON_TimeSTART : BOOL;
		T_TimeSTART : BOOL;
		T_TimeSTOP : BOOL;
		T_TimeRESET : BOOL;
		Laps_Counter_Enable : BOOL;
		Cycle_RESET : BOOL;
	END_STRUCT;
	SIKO_MASTER_Type : 	STRUCT  (* *) (* *) (*13*)
		InPosition : BOOL; (*1 - The motor is in position*) (* *) (*14*)
		PositioningInProgress : BOOL; (*1 - The positioning task is in progress*) (* *) (*15*)
		CalibrationDone : BOOL; (*1 - The calibration operation is done*) (* *) (*16*)
		MotorDisabled : BOOL; (*1 - The motor is disabled*) (* *) (*17*)
		AbortPositioning : BOOL; (*1 - The current positioning is aborted*) (* *) (*18*)
		CalibrationInProgress : BOOL; (*1 - The calibration Process is in progress*) (* *) (*19*)
		Spare_06 : BOOL; (* *) (* *) (*20*)
		Spare_07 : BOOL; (* *) (* *) (*21*)
		JogForward : BOOL; (*1 - Jog Forward Command*) (* *) (*22*)
		JogBackward : BOOL; (*1 - Jog Backward Command*) (* *) (*23*)
		StartPositioning : BOOL; (*Positive Edge - Start positioning*) (* *) (*24*)
		StartRead : BOOL; (*Positive Edge - Start read parameter from the drive*) (* *) (*25*)
		StartWrite : BOOL; (*Positive Edge - Start write parameter from the drive*) (* *) (*26*)
		Calibrate : BOOL; (*Positive Edge - Calibrate command. (Calibrate value => Current pos)*) (* *) (*27*)
		Enable : BOOL; (*0 - Disable the motor; 1 - Enable motor*) (* *) (*28*)
		Spare_17 : BOOL; (* *) (* *) (*29*)
		ReadOrWriteError : BOOL; (*1 - A read or wirte error has occured*) (* *) (*30*)
		IllegalOperation : BOOL; (*1 - An illegal operation has occurred*) (* *) (*31*)
		DeviceOutsideSwLimit : BOOL; (*1 - The device is outside the sw limit*) (* *) (*32*)
		OnError : BOOL; (*1 - The motor is on error (current, temperature too high, ...)*) (* *) (*33*)
		TargetOutsideSwLimit : BOOL; (*1 - The target position is outside the sw limit (no movement is possible)*) (* *) (*34*)
		CommunicationFault : BOOL; (*1 - Comunication fault*) (* *) (*35*)
		Spare_26 : BOOL; (* *) (* *) (*36*)
		Warning : BOOL; (*1 - Warning present*) (* *) (*37*)
		EmergencyOkFbk : BOOL; (*Emergency ok feedback*) (* *) (*38*)
		WriteEnabled : BOOL; (*1 - Write process is enabled*) (* *) (*39*)
		ReadOrWriteInProgress : BOOL; (* *) (* *) (*40*)
		Spare_33 : BOOL; (* *) (* *) (*41*)
		Spare_34 : BOOL; (* *) (* *) (*42*)
		Spare_35 : BOOL; (* *) (* *) (*43*)
		Spare_36 : BOOL; (* *) (* *) (*44*)
		Spare_37 : BOOL; (* *) (* *) (*45*)
		TargetPos : REAL; (* *) (* *) (*46*)
		CurrentPos : REAL; (* *) (* *) (*47*)
		Data : SIKO_DATA_Type; (* *) (* *) (*48*)
	END_STRUCT;
	SIKO_DATA_Type : 	STRUCT  (* *) (* *) (*50*)
		OperationMode : INT; (*r/w - address:396hex - value: 2 - Don't change!!!!!!!!!!!!!!!!!!!!!!!!!!!!!!*) (* *) (*51*)
		PGain : INT; (*r/w - address:3e8hex*) (* *) (*52*)
		IGain : INT; (*r/w - address:3e9hex*) (* *) (*53*)
		DGain : INT; (*r/w - address:3eahex*) (* *) (*54*)
		VPos : INT; (*r/w - address:3echex*) (* *) (*55*)
		APos : INT; (*r/w - address:3ebhex*) (* *) (*56*)
		VJog : INT; (*r/w - address:3f0hex*) (* *) (*57*)
		SpareInt : INT; (* *) (* *) (*58*)
		GearIn : INT; (*r/w - address:3f2hex*) (* *) (*59*)
		GearOut : INT; (*r/w - address:3f3hex*) (* *) (*60*)
		SpindlePitch : INT; (*r/w - address:3f4hex*) (* *) (*61*)
		SenseOfRotation : INT; (*r/w - address:3f5hex*) (* *) (*62*)
		UpperLimit : REAL; (*r/w - address:3f8hex*) (* *) (*63*)
		LowerLimit : REAL; (*r/w - address:3f9hex*) (* *) (*64*)
		CalibrationValue : REAL; (*r/w - address:3fahex*) (* *) (*65*)
		SystemStatusWord : INT; (*r - address:3fchex*) (* *) (*66*)
		FaultBuffer0 : UINT; (*r - address:3b1 sub: 0*) (* *) (*67*)
		FaultBuffer1 : UINT; (*r - address:3b1 sub: 1*) (* *) (*68*)
		FaultBuffer2 : UINT; (*r - address:3b1 sub: 2*) (* *) (*69*)
		FaultBuffer3 : UINT; (*r - address:3b1 sub: 3*) (* *) (*70*)
		FaultBuffer4 : UINT; (*r - address:3b1 sub: 4*) (* *) (*71*)
		FaultBuffer5 : UINT; (*r - address:3b1 sub: 5*) (* *) (*72*)
		FaultBuffer6 : UINT; (*r - address:3b1 sub: 6*) (* *) (*73*)
		FaultBuffer7 : UINT; (*r - address:3b1 sub: 7*) (* *) (*74*)
		FaultBuffer8 : UINT; (*r - address:3b1 sub: 8*) (* *) (*75*)
		FaultBuffer9 : UINT; (*r - address:3b1 sub: 9*) (* *) (*76*)
		TimeoutPositioning : TIME; (* *) (* *) (*77*)
		PosWindows : REAL; (*r/w - address:3f1hex*) (* *) (*78*)
	END_STRUCT;
	SIKO_COM_Type : 	STRUCT  (* *) (* *) (*80*)
		FLR_SIKO : FLR_SIKO_Type; (* *) (* *) (*81*)
		SIKO_FLR : SIKO_FLR_Type; (* *) (* *) (*82*)
	END_STRUCT;
	FLR_SIKO_Type : 	STRUCT  (* *) (* *) (*84*)
		PKE : UINT; (* *) (* *) (*85*)
		IND : UINT; (* *) (* *) (*86*)
		PWE_H : UINT; (* *) (* *) (*87*)
		PWE_L : UINT; (* *) (* *) (*88*)
		STW : UINT; (* *) (* *) (*89*)
		HSW_H : UINT; (* *) (* *) (*90*)
		HSW_L : UINT; (* *) (* *) (*91*)
	END_STRUCT;
	SIKO_FLR_Type : 	STRUCT  (* *) (* *) (*93*)
		PKE : UINT; (* *) (* *) (*94*)
		IND : UINT; (* *) (* *) (*95*)
		PWE_H : UINT; (* *) (* *) (*96*)
		PWE_L : UINT; (* *) (* *) (*97*)
		ZSW : UINT; (* *) (* *) (*98*)
		HIW_H : UINT; (* *) (* *) (*99*)
		HIW_L : UINT; (* *) (* *) (*100*)
	END_STRUCT;
	AlarmAreaCfg_Type : 	STRUCT  (*V4.A.A.1.6.13*)
		From : UINT;
		To : UINT;
	END_STRUCT;
	Vfd_Data_Type : 	STRUCT  (*v999_Daq*)
		Node : USINT;
		Name : STRING[80];
		ReadData : ARRAY[0..15]OF DINT;
	END_STRUCT;
END_TYPE
```

#### AlarmScheduler.st
```iecst
FUNCTION_BLOCK AlarmScheduler
	//V4.A.A.1.6.13
	memset(ADR(AlarmActionTemp), 0, SIZEOF(AlarmActionTemp));

	FOR x := 0 TO 24 DO//V1.7.2
		IF AlarmAreaCfg[x].From = 0 OR AlarmAreaCfg[x].To = 0 THEN
		ELSE
			FOR i := MAX(0, AlarmAreaCfg[x].From - 1) TO MAX(AlarmAreaCfg[x].To - 1, AlarmAreaCfg[x].From - 1) DO

				Alarm ACCESS AdrAlarm + (SIZEOF(Alarm) * i);
				AlarmCFG ACCESS AdrAlarmCFG + (SIZEOF(AlarmCFG) * i);
				AlarmOldStatus ACCESS AdrAlarmOldStatus + (SIZEOF(AlarmOldStatus) * i);
				HMI ACCESS AdrHMI + (SIZEOF(HMI) * i);

				IF FirstAlarmActive.OMAC_Index = AlarmCFG.OMAC_Index THEN
					memset(ADR(FirstAlarmActive), 0, SIZEOF(FirstAlarmActive));
				END_IF

				IF FirstExternalAlarmActive.OMAC_Index = AlarmCFG.OMAC_Index THEN
					memset(ADR(FirstExternalAlarmActive), 0, SIZEOF(FirstExternalAlarmActive));
				END_IF

				IF FirstAlarmActive.OMAC_Index = 0      AND Alarm.Active AND
					(Alarm.ActionEn AND NOT Alarm.ByPass) AND
					(AlarmCFG.Action <> 0) AND (AlarmCFG.Action <> 67) AND
					NOT Alarm.DependentActive THEN
					FirstAlarmActive := AlarmCFG;
				END_IF

				IF FirstExternalAlarmActive.OMAC_Index = 0      AND Alarm.Active AND
					(Alarm.ActionEn AND NOT Alarm.ByPass) AND
					(AlarmCFG.Action <> 0) AND (AlarmCFG.Category = 3) AND
					NOT Alarm.DependentActive THEN
					FirstExternalAlarmActive := AlarmCFG;
				END_IF

				IF Alarm.Active AND (Alarm.ActionEn AND NOT Alarm.ByPass AND Alarm.Visibility) AND
					NOT AlarmOldStatus AND NOT CriticalAcknoledgeRequest AND
					(AlarmCFG.Action > 0 AND AlarmCFG.Action < 32)	AND
					NOT Alarm.DependentActive THEN
					CriticalAcknoledgeRequest := AlarmCFG.Action <> 6; //ALARM SCHEDULER V4_03:ESCLUSIONE DEGLI ALLARMI DI SBLOCCO PORTE
				END_IF

				IF Alarm.Active AND (Alarm.ActionEn AND NOT Alarm.ByPass AND Alarm.Visibility) AND
					NOT AlarmOldStatus AND NOT AlarmAcknoledgeRequest AND
					(AlarmCFG.Action >= 32 AND AlarmCFG.Action < 64)	AND
					NOT Alarm.DependentActive THEN
					AlarmAcknoledgeRequest := TRUE;
				END_IF

				Alarm.ActionDis := NOT Alarm.ActionEn;

				HMI.0			:= Alarm.ActionEn;
				HMI.1			:= Alarm.ByPassEn;
				HMI.2;
				HMI.3;
				Alarm.ByPass	:= HMI.4;
				HMI.5			:= Alarm.ActionDis;
				HMI.6			:= Alarm.Active;
				HMI.7			:= Alarm.Visibility;

				CASE AlarmCFG.Action OF

					0:
						AlarmActionTemp.Bit.ALR_NULL					:= Alarm.Active AND NOT Alarm.DependentActive OR AlarmActionTemp.Bit.ALR_NULL;
					1:
						AlarmActionTemp.Bit.ALR_MS_QuickStop			:= Alarm.Active AND (Alarm.ActionEn AND NOT Alarm.ByPass AND NOT Alarm.DependentActive) OR AlarmActionTemp.Bit.ALR_MS_QuickStop;
					2:
						AlarmActionTemp.Bit.ALR_MS_NormalStop			:= Alarm.Active AND (Alarm.ActionEn AND NOT Alarm.ByPass AND NOT Alarm.DependentActive) OR AlarmActionTemp.Bit.ALR_MS_NormalStop;
					3:
						AlarmActionTemp.Bit.ALR_MS_QuickWithJog			:= Alarm.Active AND (Alarm.ActionEn AND NOT Alarm.ByPass AND NOT Alarm.DependentActive) OR AlarmActionTemp.Bit.ALR_MS_QuickWithJog;
					4:
						AlarmActionTemp.Bit.ALR_MS_NormalWithJog		:= Alarm.Active AND (Alarm.ActionEn AND NOT Alarm.ByPass AND NOT Alarm.DependentActive) OR AlarmActionTemp.Bit.ALR_MS_NormalWithJog;
					6:
						AlarmActionTemp.Bit.ALR_MS_NormalWithJogMnt		:= Alarm.Active AND (Alarm.ActionEn AND NOT Alarm.ByPass AND NOT Alarm.DependentActive) OR AlarmActionTemp.Bit.ALR_MS_NormalWithJogMnt;
					10:
						AlarmActionTemp.Bit.ALR_CSR_StopAfterEmptying	:= Alarm.Active AND (Alarm.ActionEn AND NOT Alarm.ByPass AND NOT Alarm.DependentActive) OR AlarmActionTemp.Bit.ALR_CSR_StopAfterEmptying;
					32:
						AlarmActionTemp.Bit.ALR_CSR						:= Alarm.Active AND (Alarm.ActionEn AND NOT Alarm.ByPass AND NOT Alarm.DependentActive) OR AlarmActionTemp.Bit.ALR_CSR;
					33:
						AlarmActionTemp.Bit.ALR_CSR_AfterSlowdown		:= Alarm.Active AND (Alarm.ActionEn AND NOT Alarm.ByPass AND NOT Alarm.DependentActive) OR AlarmActionTemp.Bit.ALR_CSR_AfterSlowdown;
					64:
						AlarmActionTemp.Bit.ALR_CSA						:= Alarm.Active AND (Alarm.ActionEn AND NOT Alarm.ByPass AND NOT Alarm.DependentActive) OR AlarmActionTemp.Bit.ALR_CSA;
					65:
						AlarmActionTemp.Bit.ALR_CSA_AfterSlowdown		:= Alarm.Active AND (Alarm.ActionEn AND NOT Alarm.ByPass AND NOT Alarm.DependentActive) OR AlarmActionTemp.Bit.ALR_CSA_AfterSlowdown;
					81:
						AlarmActionTemp.Bit.ALR_StartModeDisabled		:= Alarm.Active AND (Alarm.ActionEn AND NOT Alarm.ByPass AND NOT Alarm.DependentActive) OR AlarmActionTemp.Bit.ALR_StartModeDisabled;
					86:
						AlarmActionTemp.Bit.ALR_NoProduction			:= Alarm.Active AND (Alarm.ActionEn AND NOT Alarm.ByPass AND NOT Alarm.DependentActive) OR AlarmActionTemp.Bit.ALR_NoProduction;

					ELSE
						AlarmActionTemp.Bit.ALR_NULL					:= Alarm.Active AND NOT Alarm.DependentActive OR AlarmActionTemp.Bit.ALR_NULL;
				END_CASE

				//EXTRACTION OF FIRST ALARM FOR EACH CATEGORY
				IF FirstCriticalAlarmActive.OMAC_Index = AlarmCFG.OMAC_Index THEN//V4.A.A.1.7.0
					memset(ADR(FirstCriticalAlarmActive), 0, SIZEOF(FirstCriticalAlarmActive));
				END_IF

				IF FirstAlertAlarmActive.OMAC_Index = AlarmCFG.OMAC_Index THEN//V4.A.A.1.7.0
					memset(ADR(FirstAlertAlarmActive), 0, SIZEOF(FirstAlertAlarmActive));
				END_IF

				IF FirstExtCriticalAlarmActive.OMAC_Index = AlarmCFG.OMAC_Index THEN//V4.A.A.1.7.0
					memset(ADR(FirstExtCriticalAlarmActive), 0, SIZEOF(FirstExtCriticalAlarmActive));
				END_IF

				IF FirstExtAlertAlarmActive.OMAC_Index = AlarmCFG.OMAC_Index THEN//V4.A.A.1.7.0
					memset(ADR(FirstExtAlertAlarmActive), 0, SIZEOF(FirstExtAlertAlarmActive));
				END_IF
				IF FirstCsAlarmActive.OMAC_Index = AlarmCFG.OMAC_Index THEN//V4.A.A.1.7.0
					memset(ADR(FirstCsAlarmActive), 0, SIZEOF(FirstCsAlarmActive));
				END_IF
				//V4.A.A.1.7.0
				IF FirstCriticalAlarmActive.OMAC_Index = 0	AND Alarm.Active		AND
					(Alarm.ActionEn					AND NOT Alarm.ByPass)		AND
					(AlarmCFG.Action > 0)			AND (AlarmCFG.Action <= 31)	AND (AlarmCFG.Category <> 3) AND
					NOT Alarm.DependentActive THEN
					FirstCriticalAlarmActive := AlarmCFG;
				END_IF
				//V4.A.A.1.7.0
				IF FirstAlertAlarmActive.OMAC_Index = 0	AND Alarm.Active			AND
					(Alarm.ActionEn					AND NOT Alarm.ByPass)		AND
					(AlarmCFG.Action >= 32)			AND (AlarmCFG.Action <= 63)	AND (AlarmCFG.Category <> 3) AND
					NOT Alarm.DependentActive THEN
					FirstAlertAlarmActive := AlarmCFG;
				END_IF
				//V4.A.A.1.7.5a
				IF FirstCsAlarmActive.OMAC_Index = 0	AND Alarm.Active			AND
					(Alarm.ActionEn							AND NOT Alarm.ByPass)		AND
					(AlarmCFG.Action >= 64)			AND (AlarmCFG.Action <= 65) AND (AlarmCFG.Category <> 3)	AND
					NOT Alarm.DependentActive THEN
					FirstCsAlarmActive := AlarmCFG;
				END_IF
				//V4.A.A.1.7.0
				IF FirstExtCriticalAlarmActive.OMAC_Index = 0	AND Alarm.Active			AND
					(Alarm.ActionEn							AND NOT Alarm.ByPass)		AND
					(AlarmCFG.Action > 0)			AND (AlarmCFG.Action <= 31)	AND (AlarmCFG.Category = 3)	AND
					NOT Alarm.DependentActive THEN
					FirstExtCriticalAlarmActive := AlarmCFG;
				END_IF
				//V4.A.A.1.7.0
				IF FirstExtAlertAlarmActive.OMAC_Index = 0	AND Alarm.Active			AND
					(Alarm.ActionEn							AND NOT Alarm.ByPass)		AND
					(AlarmCFG.Action >= 32)			AND (AlarmCFG.Action <= 63)	AND (AlarmCFG.Category = 3)	AND
					NOT Alarm.DependentActive THEN
					FirstExtAlertAlarmActive := AlarmCFG;
				END_IF
				//V4.A.A.1.7.5a
				IF FirstCsAlarmActive.OMAC_Index = 0	AND Alarm.Active			AND
					(Alarm.ActionEn							AND NOT Alarm.ByPass)		AND
					(AlarmCFG.Action >= 64)			AND (AlarmCFG.Action <= 65)	AND (AlarmCFG.Category = 3)	AND
					NOT Alarm.DependentActive THEN
					FirstCsExtAlarmActive := AlarmCFG;
				END_IF
				//END EXTRACTION

				AlarmOldStatus := Alarm.Active AND (Alarm.ActionEn AND NOT Alarm.ByPass AND NOT Alarm.DependentActive);
			END_FOR
		END_IF
	END_FOR

	AlarmAction	:= AlarmActionTemp;
END_FUNCTION_BLOCK

FUNCTION_BLOCK FirstAlarmCombiner
	IF (FirstAlarmActive.OMAC_Index >= SkidAlarmFrom) AND (FirstAlarmActive.OMAC_Index <= SkidAlarmTo) THEN
		memset(ADR(FirstAlarmActive), 0, SIZEOF(FirstAlarmActive));
	END_IF

	IF (FirstExternalAlarmActive.OMAC_Index >= SkidAlarmFrom) AND (FirstExternalAlarmActive.OMAC_Index <= SkidAlarmTo) THEN
		memset(ADR(FirstExternalAlarmActive), 0, SIZEOF(FirstExternalAlarmActive));
	END_IF

	IF SkidFirstAlarm <> 0 AND FirstAlarmActive.OMAC_Index = 0 THEN
		FirstAlarmActive.OMAC_Index := SkidFirstAlarm;
		AlarmCFG ACCESS AdrAlarmCFG + (SIZEOF(AlarmCFG) * SkidFirstAlarm);
		FirstAlarmActive.OMAC_Code	:= AlarmCFG.OMAC_Code; //V1.7.4
	END_IF

	IF SkidFirstExternalAlarm <> 0 AND FirstExternalAlarmActive.OMAC_Index = 0 THEN
		FirstExternalAlarmActive.OMAC_Index := SkidFirstExternalAlarm;
		AlarmCFG ACCESS AdrAlarmCFG + (SIZEOF(AlarmCFG) * SkidFirstExternalAlarm);
		FirstExternalAlarmActive.OMAC_Code 	:= AlarmCFG.OMAC_Code;//V1.7.4
	END_IF
END_FUNCTION_BLOCK
```

#### AnalogTotalizer.st
```iecst
FUNCTION_BLOCK AnalogTotalizer
	RTInfo(enable := TRUE);

	CASE IN_ConfigType OF
		0:
			VAR_AuxPulse := IN_PulseWeight * BOOL_TO_REAL(EDGEPOS(IN_Pulse));
		1:
			VAR_AuxPulse := IN_AnalogPV * UDINT_TO_REAL(RTInfo.cycle_time) /1000000;
		2:
			VAR_AuxPulse := IN_AnalogPV * UDINT_TO_REAL(RTInfo.cycle_time) /1000000 / 60;
		3:
			VAR_AuxPulse := IN_AnalogPV * UDINT_TO_REAL(RTInfo.cycle_time) /1000000 / 3600;
	END_CASE

	OUT_TotalCounter := VAR_AuxPulse + OUT_TotalCounter;

	IF IN_Reset THEN
		OUT_TotalCounter := 0.0;
	END_IF
END_FUNCTION_BLOCK
```

#### Blink.st
```iecst
FUNCTION_BLOCK FB_Blinker
	VAR_TimeValue	:= REAL_TO_TIME((1.0 / IN_Freq) * 1000);

	TMR_TON_OnDelay(IN:= NOT OUT,	PT:= VAR_TimeValue / 2);
	TMR_TON_OffDelay(IN:= OUT,		PT:= VAR_TimeValue / 2);

	IF TMR_TON_OnDelay.Q THEN
		OUT	:= TRUE;
	ELSIF TMR_TON_OffDelay.Q THEN
		OUT	:= FALSE;
	END_IF
END_FUNCTION_BLOCK
```

#### ComboBox.st
```iecst
FUNCTION ComboBoxString
	OUT_ComboString := '';
	FOR VAR_ElementsIndex := 0 TO 19 DO
		IF IN_ElementsStructure[VAR_ElementsIndex].Present THEN
			itoa(USINT_TO_DINT(VAR_ElementsIndex), ADR(VAR_StrIndex));
			VAR_StrComma 		:= ',';
			VAR_StrSemicolun 	:= ';';
			strcat(ADR(OUT_ComboString), ADR(VAR_StrIndex));
			strcat(ADR(OUT_ComboString), ADR(VAR_StrComma));
			strcat(ADR(OUT_ComboString), ADR(IN_ElementsStructure[VAR_ElementsIndex].Name));
			strcat(ADR(OUT_ComboString), ADR(VAR_StrSemicolun));
		END_IF
	END_FOR
	ComboBoxString := TRUE;
END_FUNCTION
```

#### CyclicActivation.st
```iecst
FUNCTION_BLOCK CyclicActivation
	VAR_RtInfo(enable:=TRUE);
	VAR_CycleCounter	:= MAX(1, VAR_CycleCounter + 1);
	OUT_A	:= FALSE;
	OUT_B	:= FALSE;

	TMR_TON_CycleA(	IN := VAR_Cycle,
	PT := (IN_CycleTime / 2) - UDINT_TO_TIME(VAR_RtInfo.cycle_time / 1000));

	TMR_TON_CycleB(	IN := NOT VAR_Cycle,
	PT := (IN_CycleTime / 2) - UDINT_TO_TIME(VAR_RtInfo.cycle_time / 1000));

	IF TMR_TON_CycleA.Q THEN
		OUT_A		:= TRUE;
		VAR_Cycle	:= FALSE;
	ELSIF TMR_TON_CycleB.Q THEN
		OUT_B		:= TRUE;
		VAR_Cycle	:= TRUE;
	ELSE
		RETURN;
	END_IF

	VAR_CycleTime	:= (UDINT_TO_REAL(VAR_RtInfo.cycle_time) * VAR_CycleCounter) / 1000000.0;
	VAR_CycleCounter 	:= 0.0;
	memset(ADR(TMR_TON_CycleA), 0, SIZEOF(TMR_TON_CycleA));
	memset(ADR(TMR_TON_CycleB), 0, SIZEOF(TMR_TON_CycleB));
END_FUNCTION_BLOCK
```
